DATA_BLOCK "Inputs"   // DB13
{ S7_Optimized_Access := 'FALSE' }
VERSION : 0.1
   VAR
      "BC01 run" : Bool;
      BC01_All_inv : Bool;
      "RD01 run" : Bool;
      RD01_All_inv : Bool;
      "fan RD01 run" : Bool;
      "MC03 run" : Bool;
      "MC04 run" : Bool;
      MC04_All_inv : Bool;
      "MC05 run" : Bool;
      "VS01 run" : Bool;
      VS01_All_Inv : Bool;
      "FEEDBACKMOTOR SC-12" : Bool;
      "Aux inverter RUN" : Bool;
      Aux_Inv_All : Bool;
      "MV06 Run_Opening" : Bool;
      "MV06 Run_Closing" : Bool;
      "MV05 RUN_Opening" : Bool;
      "MV05 RUN_Closing" : Bool;
      "MV02 RUN_Opening" : Bool;
      "MV02 RUN_Closing" : Bool;
      "MV03 Run_Opening" : Bool;
      "MV03 Run_Closing" : Bool;
      "MV04 RUN_Opening" : Bool;
      "MV04 RUN_Closing" : Bool;
      "FN02 Run" : Bool;
      FN02_All_Inv : Bool;
      "MV01 Run_Opening" : Bool;
      "MV01 Run_Closing" : Bool;
      "VR-01 RUN" : Bool;
      "FN01 Run" : Bool;
      FN01_All_Inv : Bool;
      "VR02 Run" : Bool;
      "CH01 Run" : Bool;
      "FN03 Run" : Bool;
      FN03_All_SoftStarter : Bool;
      "FEEDBACKMOTOR FN-06" : Bool;
      "FEEDBACKMOTOR SC-01" : Bool;
      "FEEDBACKMOTOR FN-01 FAN" : Bool;
      "FEEDBACKMOTOR LD-01" : Bool;
      "FEEDBACKMOTOR-LD-01A" : Bool;
      "FEEDBACKMOTOR SC-10" : Bool;
      "FEEDBACKMOTOR SC-11" : Bool;
      SPARE_0 : Bool;
      SPARE_1 : Bool;
      "VR03 Run" : Bool;
      "VR04 Run" : Bool;
      "VR05 Run" : Bool;
      "VR-06 RUN" : Bool;
      "FN-05 RUN" : Bool;
      Feedback_ER01 : Bool;
      "BC01 trip wire" : Bool;
      "BC01 prox" : Bool;
      "MC03 torque" : Bool;
      "MC04 torque" : Bool;
      "MC05 torque" : Bool;
      MV06_Open : Bool;
      "MV06 Close" : Bool;
      "MV05 open" : Bool;
      "MV05 Close" : Bool;
      "MV02 Open" : Bool;
      "MV02 Close" : Bool;
      "MV03 open" : Bool;
      "MV03 Close" : Bool;
      "MV04 Open" : Bool;
      "MV04 Close" : Bool;
      "MV01 Open" : Bool;
      "MV01 Close" : Bool;
      SPARE_2 : Bool;
      SPARE_3 : Bool;
      SPARE_4 : Bool;
      "FC GATE A OPEN" : Bool;
      "LIMIT SWITCH LS-02GATE A CLOSEDVALVE PV-01" : Bool;
      "PV-01 GATE B OPEN" : Bool;
      "LIMIT SWITCH LS-06GATE B CLOSEDVALVE PV-01" : Bool;
      "Selector Op Gate A PV-01" : Bool;
      "Selector Op Gate B PV-01" : Bool;
      "PV-02 EV A OPEN" : Bool;
      "PV-02 EV A CLOSE" : Bool;
      "PV-02 GATE B OPEN" : Bool;
      "PV-02 GATE B CLOSE" : Bool;
      "Selector Op Gate A PV-02" : Bool;
      "Selector Op Gate B PV-02" : Bool;
      "Deviator Open PV-03" : Bool;
      "Deviator Close PV-03" : Bool;
      "PV03 Local Selector" : Bool;
      "PV04 Open" : Bool;
      "PV04 Close" : Bool;
      "Button Open PV-0000" : Bool;
      "Low Pressure Air" : Bool;
      "BWF01 OK" : Bool;
      "BWF 01 RUN" : Bool;
      "BWF01 FAULT" : Bool;
      "min LEV BWF01" : Bool;
      "MAX LEV BWF01" : Bool;
      "BWF02 OK" : Bool;
      "BWF 02 RUN" : Bool;
      "BWF02 FAULT" : Bool;
      "min LEV BWF02" : Bool;
      "MAX LEV BWF02" : Bool;
      "APRON CONVEYOR A RUN" : Bool;
      "IMPACTOR RUN" : Bool;
      "IMPACT VIBRATIONFEEDER RUN" : Bool;
      "BELT CONVEYOR A RUN" : Bool;
      "AIR KNIFE RUN" : Bool;
      "BELT CONVEYOR B RUN" : Bool;
      "SHREDDER 1 RUN" : Bool;
      "SHREDDER VIBRATIONFEEDER RUN" : Bool;
      "BELT CONVEYOR  C RUN" : Bool;
      "ROTEX SCREEN RUN" : Bool;
      "APRON CONVEYOR B RUN" : Bool;
      "SHREDDER 2 RUN" : Bool;
      "BELT CONVEYOR  D RUN" : Bool;
      "BELT CONVEYOR E RUN" : Bool;
      "LIW SYSTEMAUTOREADER" : Bool;
      "PRIMARYSHREDDER RUN" : Bool;
      FREE : Bool;
      BWF1_INVERTER_HIGH_SPEED : Bool;
      BWF2_INVERTER_HIGH_SPEED : Bool;
      "APRON CONVEYOR A FAULT" : Bool;
      "IMPACTOR FAULT" : Bool;
      "IMPACT VIBRATIONFEEDER FAULT" : Bool;
      "BELT CONVEYOR  A FAULT" : Bool;
      "AIR KNIFE FAULT" : Bool;
      "BELT CONVEYOR B FAULT" : Bool;
      "SHREDDER 1 FAULT" : Bool;
      "SHREDDER VIBRATIONFEEDER FAULT" : Bool;
      "BELT CONVEYOR C FAULT" : Bool;
      "ROTEX SCREENFAULT" : Bool;
      "APRON CONVEYOR B FAULT" : Bool;
      "SHREDDER 2FAULT" : Bool;
      "BELT COVEYOR  D FAULT" : Bool;
      "BELT CONVEYOR  E FAULT" : Bool;
      "WEIGHTING HOPPER 2FAULT" : Bool;
      "HOPPER CONVEYOR 2FAULT" : Bool;
      "BELT CONVEYOR C FAULT_doppio!" : Bool;
      "NITROGEN TANK READY" : Bool;
      "Burner On" : Bool;
      "Brurner Lock Out" : Bool;
      "Burner ON and OK" : Bool;
      "FC GAS Chiuso" : Bool;
      "Max Pressure Gas" : Bool;
      "FC Aria chiusa" : Bool;
      "FC Aria aperta" : Bool;
      "High Flame Gas" : Bool;
      FREE_2 : Bool;
      FREE_3 : Bool;
      FREE_4 : Bool;
      FREE_5 : Bool;
      FREE_6 : Bool;
      FREE_7 : Bool;
      FREE_8 : Bool;
      FREE_9 : Bool;
      FREE_10 : Bool;
      FREE_11 : Bool;
      FREE_12 : Bool;
      FREE_13 : Bool;
      EM_OK : Bool;
      Presenza_110V : Bool;
      Tacitazione : Bool;
      Reset_allarmi : Bool;
      MV01_CHANNEL_D : Bool;
      MV01_CHANNEL_C : Bool;
      MV02_CHANNEL_D : Bool;
      MV02_CHANNEL_C : Bool;
      MV03_CHANNEL_D : Bool;
      MV03_CHANNEL_C : Bool;
      MV05_CHANNEL_D : Bool;
      MV05_CHANNEL_C : Bool;
      MV06_CHANNEL_D : Bool;
      MV06_CHANNEL_C : Bool;
      FREE_23 : Bool;
      FREE_24 : Bool;
      FREE_25 : Bool;
      FREE_26 : Bool;
      FREE_27 : Bool;
      FREE_28 : Bool;
      "PV-14 OPEN" : Bool;
      "PV-14 CLOSE" : Bool;
      "FN04 Run" : Bool;
      FN04_All_inv : Bool;
      "177T1_OK" : Bool;
      "LD-01 Minimo" : Bool;
      "LD-01 Inspection LS" : Bool;
      "LD-01 Local Button" : Bool;
      TC_04 : Word;
      TC_05 : Word;
      Flow_rate_BWF01 : Word;
      Flow_rate_BWF02 : Word;
      Level_BWF01 : Word;
      Level_BWF02 : Word;
      TC_01 : Word;
      TC_02 : Word;
      TC_03 : Word;
      TC_06 : Word;
      TC_07 : Word;
      ZT_01 : Word;
      PSH_01 : Word;
      PSH_02 : Word;
      PSH_03 : Word;
      PC_01 : Word;
      MV_04_M18A : Word;
      MV_04_MV18B : Word;
      FN02_ABSORPTION : Word;
      FN04_ABSORPTION : Word;
      RD01_ABSORBPTION : Word;
      FN01_ABSORPTION : Word;
      RO_01 : Word;
      RO_02 : Word;
      RO_03 : Word;
      RO_04 : Word;
      BR_01_RETRANSMISSION_GAS : Word;
      BR_01_RETRANSMISSION_AIR : Word;
      BR_01_MASSFLOWMETER_GAS : Word;
      BR_01_MASSFLOWMETER_AIR : Word;
   END_VAR
BEGIN
END_DATA_BLOCK

DATA_BLOCK "Output"   // DB14
{ S7_Optimized_Access := 'FALSE' }
VERSION : 0.1
   VAR
      "Start BC01" : Bool;
      "Start RD01" : Bool;
      "Start fan RD01" : Bool;
      "Start Spare Motor" : Bool;
      "Start MC04" : Bool;
      "Start MC05" : Bool;
      "Start VS01" : Bool;
      "Start SC12" : Bool;
      "Start Aux INV" : Bool;
      "Open MV06" : Bool;
      "Close MV06" : Bool;
      "Open MV05" : Bool;
      "Close MV05" : Bool;
      "Open MV02" : Bool;
      "Close MV02" : Bool;
      "Start open MV03" : Bool;
      "Start Close MV03" : Bool;
      "Open MV04" : Bool;
      "Close MV04" : Bool;
      "Start FN02" : Bool;
      "Start Open MV-01" : Bool;
      "Start Close MV-01" : Bool;
      "Start VR01" : Bool;
      "Start FN01" : Bool;
      "Start VR02" : Bool;
      "Start CH01" : Bool;
      "Start FN03" : Bool;
      "Start FN06" : Bool;
      "Start SC01" : Bool;
      "Star fan FN01" : Bool;
      "Start LD01" : Bool;
      "Start Vibrator LD-01" : Bool;
      "Start SC10" : Bool;
      "Start SC11" : Bool;
      "Start FN04" : Bool;
      "Start VR03" : Bool;
      "Start VR04" : Bool;
      "Start VR05" : Bool;
      "Start VR06" : Bool;
      "Start FN05" : Bool;
      "Start ER-01" : Bool;
      EV03 : Bool;
      "PV-01 Gate a" : Bool;
      "PV-01 GATE B EV" : Bool;
      "PV-02 GATE A EV" : Bool;
      "PV-02 GATE B EV" : Bool;
      "PV-03 GATE EV" : Bool;
      "PV-04" : Bool;
      "Abilita start chiller" : Bool;
      "START LIW FEEDER" : Bool;
      "Consenso Start BWF01" : Bool;
      "Consenso Start BWF02" : Bool;
      "Start Nitrogen" : Bool;
      "Rem. Start/Stop Burner" : Bool;
      "Temperature Interlock OK" : Bool;
      "Rst allarm Burner" : Bool;
      "Start High Flame" : Bool;
      "Forzatura scintilla" : Bool;
      Spare_30 : Bool;
      Spare_31 : Bool;
      Spare_32 : Bool;
      Spare_33 : Bool;
      Siren : Bool;
      "Blinking Ligh" : Bool;
      Spare : Bool;
      Spare_1 : Bool;
      Spare_2 : Bool;
      Spare_3 : Bool;
      Spare_4 : Bool;
      Spare_5 : Bool;
      Spare_6 : Bool;
      Spare_7 : Bool;
      Spare_8 : Bool;
      Spare_9 : Bool;
      Spare_10 : Bool;
      Spare_11 : Bool;
      Spare_12 : Bool;
      Spare_13 : Bool;
      Spare_14 : Bool;
      Spare_15 : Bool;
      Spare_16 : Bool;
      Spare_17 : Bool;
      Spare_18 : Bool;
      Spare_19 : Bool;
      Spare_20 : Bool;
      Spare_21 : Bool;
      Spare_22 : Bool;
      Spare_23 : Bool;
      Spare_24 : Bool;
      Spare_25 : Bool;
      Spare_26 : Bool;
      Spare_27 : Bool;
      Spare_28 : Bool;
      Spare_29 : Bool;
      Spare_34 : Bool;
      Spare_35 : Bool;
      "EV-11" : Bool;
      "EV-12" : Bool;
      "EV-13" : Bool;
      "EV-14" : Bool;
      "EV-15" : Bool;
      "EV-16" : Bool;
      "EV-17" : Bool;
      "EV-18" : Bool;
      "EV-19" : Bool;
      "EV-20" : Bool;
      "EV-21" : Bool;
      "EV-22" : Bool;
      "EV-23" : Bool;
      "EV-24" : Bool;
      "EV-25" : Bool;
      "EV-26" : Bool;
      "EV-27" : Bool;
      "EV-28" : Bool;
      "EV-29" : Bool;
      "EV-30" : Bool;
      "EV-31" : Bool;
      "EV-32" : Bool;
      "EV-33" : Bool;
      "EV-34" : Bool;
      "EV-35" : Bool;
      "EV-36" : Bool;
      "EV-37" : Bool;
      "EV-38" : Bool;
      "EV-39" : Bool;
      "EV-40" : Bool;
      "EV-41" : Bool;
      "EV-42" : Bool;
      "EV-43" : Bool;
      "EV-44" : Bool;
      "EV-45" : Bool;
      "EV-46" : Bool;
      "EV-47" : Bool;
      "EV-48" : Bool;
      "EV-49" : Bool;
      "EV-50" : Bool;
      "PV-14" : Bool;
      Spare_36 : Bool;
      Spare_37 : Bool;
      Spare_38 : Bool;
      Spare_39 : Bool;
      Spare_40 : Bool;
      Spare_41 : Bool;
      Spare_42 : Bool;
      "EV-51" : Bool;
      "EV-52" : Bool;
      "EV-53" : Bool;
      "EV-54" : Bool;
      "EV-55" : Bool;
      "EV-56" : Bool;
      "EV-57" : Bool;
      "EV-58" : Bool;
      "EV-59" : Bool;
      "EV-60" : Bool;
      "EV- 61" : Bool;
      "EV-62" : Bool;
      "EV-63" : Bool;
      "EV-64" : Bool;
      "EV-65" : Bool;
      "EV-66" : Bool;
      "EV-67" : Bool;
      "EV-68" : Bool;
      "EV-69" : Bool;
      "EV-70" : Bool;
      "EV-71" : Bool;
      "EV-72" : Bool;
      "EV-73" : Bool;
      "EV-74" : Bool;
      "EV-75" : Bool;
      "EV-76" : Bool;
      "EV-77" : Bool;
      "EV-78" : Bool;
      "EV-79" : Bool;
      "EV-80" : Bool;
      "EV-81" : Bool;
      "EV-82" : Bool;
      "EV-83" : Bool;
      "EV-84" : Bool;
      "EV-85" : Bool;
      "EV- 86" : Bool;
      "EV-87" : Bool;
      "EV-88" : Bool;
      "EV-89" : Bool;
      "EV-90" : Bool;
   END_VAR
BEGIN
END_DATA_BLOCK

DATA_BLOCK "RecipesDB"   // DB26
{ S7_Optimized_Access := 'FALSE' }
VERSION : 0.1
   VAR
      HMI_Index : Int;   // Recipe Currently Displayed on Editor (1...100)
      OldHmi_Idx : Int;   // Last Scan Hmi idx
      Vis_SaveUndo : Bool;   // Vsibility For Undo and Save btn
      Vis_Modify : Bool := 1;   // Vsibility For Modify btn
      Vis_LoadRecipe : Bool := 1;   // Visibility Of the load recipe btn
      Load_Recipe : Bool;   // Load Recipe In Cycle
      Save_Recipe : Bool;   // Save Recipe in Archive
      Modify_Recipe : Bool;   // Modify The Editor Displayed Recipe
      Undo_Modification : Bool;   // Undo the edits on the editor
      Active_Recipe : Int;   // Recipe Currently Used
      Recipes : Array[0..101] of "Recipe";   // 100 Records Of recipes + HMI Buffer
   END_VAR
BEGIN
   // Recipes[0] : HMI Buffer
   // Recipes[1] : Recipe #1
   // Recipes[2] : Recipe #2
   // Recipes[3] : Recipe #3
   // Recipes[4] : Recipe #4
   // Recipes[5] : Recipe #5
   // Recipes[6] : Recipe #6
   // Recipes[7] : Recipe #7
   // Recipes[8] : Recipe #8
   // Recipes[9] : Recipe #9
   // Recipes[10] : Recipe #10
   // Recipes[11] : Recipe #11
   // Recipes[12] : Recipe #12
   // Recipes[13] : Recipe #13
   // Recipes[14] : Recipe #14
   // Recipes[15] : Recipe #15
   // Recipes[16] : Recipe #16
   // Recipes[17] : Recipe #17
   // Recipes[18] : Recipe #18
   // Recipes[19] : Recipe #19
   // Recipes[20] : Recipe #20
   // Recipes[21] : Recipe #21
   // Recipes[22] : Recipe #22
   // Recipes[23] : Recipe #23
   // Recipes[24] : Recipe #24
   // Recipes[25] : Recipe #25
   // Recipes[26] : Recipe #26
   // Recipes[27] : Recipe #27
   // Recipes[28] : Recipe #28
   // Recipes[29] : Recipe #29
   // Recipes[30] : Recipe #30
   // Recipes[31] : Recipe #31
   // Recipes[32] : Recipe #32
   // Recipes[33] : Recipe #33
   // Recipes[34] : Recipe #34
   // Recipes[35] : Recipe #35
   // Recipes[36] : Recipe #36
   // Recipes[37] : Recipe #37
   // Recipes[38] : Recipe #38
   // Recipes[39] : Recipe #39
   // Recipes[40] : Recipe #40
   // Recipes[41] : Recipe #41
   // Recipes[42] : Recipe #42
   // Recipes[43] : Recipe #43
   // Recipes[44] : Recipe #44
   // Recipes[45] : Recipe #45
   // Recipes[46] : Recipe #46
   // Recipes[47] : Recipe #47
   // Recipes[48] : Recipe #48
   // Recipes[49] : Recipe #49
   // Recipes[50] : Recipe #50
   // Recipes[51] : Recipe #51
   // Recipes[52] : Recipe #52
   // Recipes[53] : Recipe #53
   // Recipes[54] : Recipe #54
   // Recipes[55] : Recipe #55
   // Recipes[56] : Recipe #56
   // Recipes[57] : Recipe #57
   // Recipes[58] : Recipe #58
   // Recipes[59] : Recipe #59
   // Recipes[60] : Recipe #60
   // Recipes[61] : Recipe #61
   // Recipes[62] : Recipe #62
   // Recipes[63] : Recipe #63
   // Recipes[64] : Recipe #64
   // Recipes[65] : Recipe #65
   // Recipes[66] : Recipe #66
   // Recipes[67] : Recipe #67
   // Recipes[68] : Recipe #68
   // Recipes[69] : Recipe #69
   // Recipes[70] : Recipe #70
   // Recipes[71] : Recipe #71
   // Recipes[72] : Recipe #72
   // Recipes[73] : Recipe #73
   // Recipes[74] : Recipe #74
   // Recipes[75] : Recipe #75
   // Recipes[76] : Recipe #76
   // Recipes[77] : Recipe #77
   // Recipes[78] : Recipe #78
   // Recipes[79] : Recipe #79
   // Recipes[80] : Recipe #80
   // Recipes[81] : Recipe #81
   // Recipes[82] : Recipe #82
   // Recipes[83] : Recipe #83
   // Recipes[84] : Recipe #84
   // Recipes[85] : Recipe #85
   // Recipes[86] : Recipe #86
   // Recipes[87] : Recipe #87
   // Recipes[88] : Recipe #88
   // Recipes[89] : Recipe #89
   // Recipes[90] : Recipe #90
   // Recipes[91] : Recipe #91
   // Recipes[92] : Recipe #92
   // Recipes[93] : Recipe #93
   // Recipes[94] : Recipe #94
   // Recipes[95] : Recipe #95
   // Recipes[96] : Recipe #96
   // Recipes[97] : Recipe #97
   // Recipes[98] : Recipe #98
   // Recipes[99] : Recipe #99
   // Recipes[100] : Recipe #100
END_DATA_BLOCK

// folder: System blocks/Program resources

DATA_BLOCK "Clock1S_simu"   // DB28
{ S7_Optimized_Access := 'TRUE' }
AUTHOR : Simatic
FAMILY : IEC
NAME : IEC_TMR
VERSION : 1.0
// stored: InstanceOfName IEC_TIMER
"IEC_TIMER"
BEGIN
END_DATA_BLOCK

DATA_BLOCK "Clock3s_simu"   // DB29
{ S7_Optimized_Access := 'TRUE' }
AUTHOR : Simatic
FAMILY : IEC
NAME : IEC_TMR
VERSION : 1.0
// stored: InstanceOfName IEC_TIMER
"IEC_TIMER"
BEGIN
END_DATA_BLOCK

DATA_BLOCK "Aux_Inv_run"   // DB31
{ S7_Optimized_Access := 'TRUE' }
AUTHOR : Simatic
FAMILY : IEC
NAME : IEC_TMR
VERSION : 1.0
// stored: InstanceOfName IEC_TIMER
"IEC_TIMER"
BEGIN
END_DATA_BLOCK

DATA_BLOCK "Er_01_Run_Rit"   // DB32
{ S7_Optimized_Access := 'TRUE' }
AUTHOR : Simatic
FAMILY : IEC
NAME : IEC_TMR
VERSION : 1.0
// stored: InstanceOfName IEC_TIMER
"IEC_TIMER"
BEGIN
END_DATA_BLOCK

DATA_BLOCK "Min_LD_01"   // DB33
{ S7_Optimized_Access := 'TRUE' }
AUTHOR : Simatic
FAMILY : IEC
NAME : IEC_TMR
VERSION : 1.0
// stored: InstanceOfName IEC_TIMER
"IEC_TIMER"
BEGIN
END_DATA_BLOCK

DATA_BLOCK "RO03_Min"   // DB34
{ S7_Optimized_Access := 'TRUE' }
AUTHOR : Simatic
FAMILY : IEC
NAME : IEC_TMR
VERSION : 1.0
// stored: InstanceOfName IEC_TIMER
"IEC_TIMER"
BEGIN
END_DATA_BLOCK

DATA_BLOCK "RO03_Max"   // DB35
{ S7_Optimized_Access := 'TRUE' }
AUTHOR : Simatic
FAMILY : IEC
NAME : IEC_TMR
VERSION : 1.0
// stored: InstanceOfName IEC_TIMER
"IEC_TIMER"
BEGIN
END_DATA_BLOCK

DATA_BLOCK "IEC_Timer_0_DB"   // DB36
{ S7_Optimized_Access := 'TRUE' }
AUTHOR : Simatic
FAMILY : IEC
NAME : IEC_TMR
VERSION : 1.0
// stored: InstanceOfName IEC_TIMER
"IEC_TIMER"
BEGIN
END_DATA_BLOCK

DATA_BLOCK "IEC_Timer_1_DB"   // DB37
{ S7_Optimized_Access := 'TRUE' }
AUTHOR : Simatic
FAMILY : IEC
NAME : IEC_TMR
VERSION : 1.0
// stored: InstanceOfName IEC_TIMER
"IEC_TIMER"
BEGIN
END_DATA_BLOCK

DATA_BLOCK "T_Reset_Startup_PV1"   // DB38
{ S7_Optimized_Access := 'TRUE' }
AUTHOR : Simatic
FAMILY : IEC
NAME : IEC_TMR
VERSION : 1.0
// stored: InstanceOfName IEC_TIMER
"IEC_TIMER"
BEGIN
END_DATA_BLOCK

DATA_BLOCK "ton_1st_step_FN01"   // DB42
{ S7_Optimized_Access := 'TRUE' }
AUTHOR : Simatic
FAMILY : IEC
NAME : IEC_TMR
VERSION : 1.0
// stored: InstanceOfName IEC_TIMER
"IEC_TIMER"
BEGIN
END_DATA_BLOCK

DATA_BLOCK "ton_2nd_step_FN01"   // DB43
{ S7_Optimized_Access := 'TRUE' }
AUTHOR : Simatic
FAMILY : IEC
NAME : IEC_TMR
VERSION : 1.0
// stored: InstanceOfName IEC_TIMER
"IEC_TIMER"
BEGIN
END_DATA_BLOCK

DATA_BLOCK "ton_3rd_step_FN01"   // DB44
{ S7_Optimized_Access := 'TRUE' }
AUTHOR : Simatic
FAMILY : IEC
NAME : IEC_TMR
VERSION : 1.0
// stored: InstanceOfName IEC_TIMER
"IEC_TIMER"
BEGIN
END_DATA_BLOCK

DATA_BLOCK "ton_4th_step_FN01"   // DB45
{ S7_Optimized_Access := 'TRUE' }
AUTHOR : Simatic
FAMILY : IEC
NAME : IEC_TMR
VERSION : 1.0
// stored: InstanceOfName IEC_TIMER
"IEC_TIMER"
BEGIN
END_DATA_BLOCK

DATA_BLOCK "ton_last_step_FN01"   // DB46
{ S7_Optimized_Access := 'TRUE' }
AUTHOR : Simatic
FAMILY : IEC
NAME : IEC_TMR
VERSION : 1.0
// stored: InstanceOfName IEC_TIMER
"IEC_TIMER"
BEGIN
END_DATA_BLOCK

DATA_BLOCK "IEC_Timer_0_DB_1"   // DB47
{ S7_Optimized_Access := 'TRUE' }
AUTHOR : Simatic
FAMILY : IEC
NAME : IEC_TMR
VERSION : 1.0
// stored: InstanceOfName IEC_TIMER
"IEC_TIMER"
BEGIN
END_DATA_BLOCK

// folder: (top level)

FUNCTION "time work motor" : Void   // FC2, LAD
{ S7_Optimized_Access := 'FALSE' }
VERSION : 0.1
   VAR_TEMP   // added for the SCL form of the ladder/FBD networks
      _w1 : Bool;
      _w2 : Bool;
   END_VAR
BEGIN

REGION Network 1: client motor 1
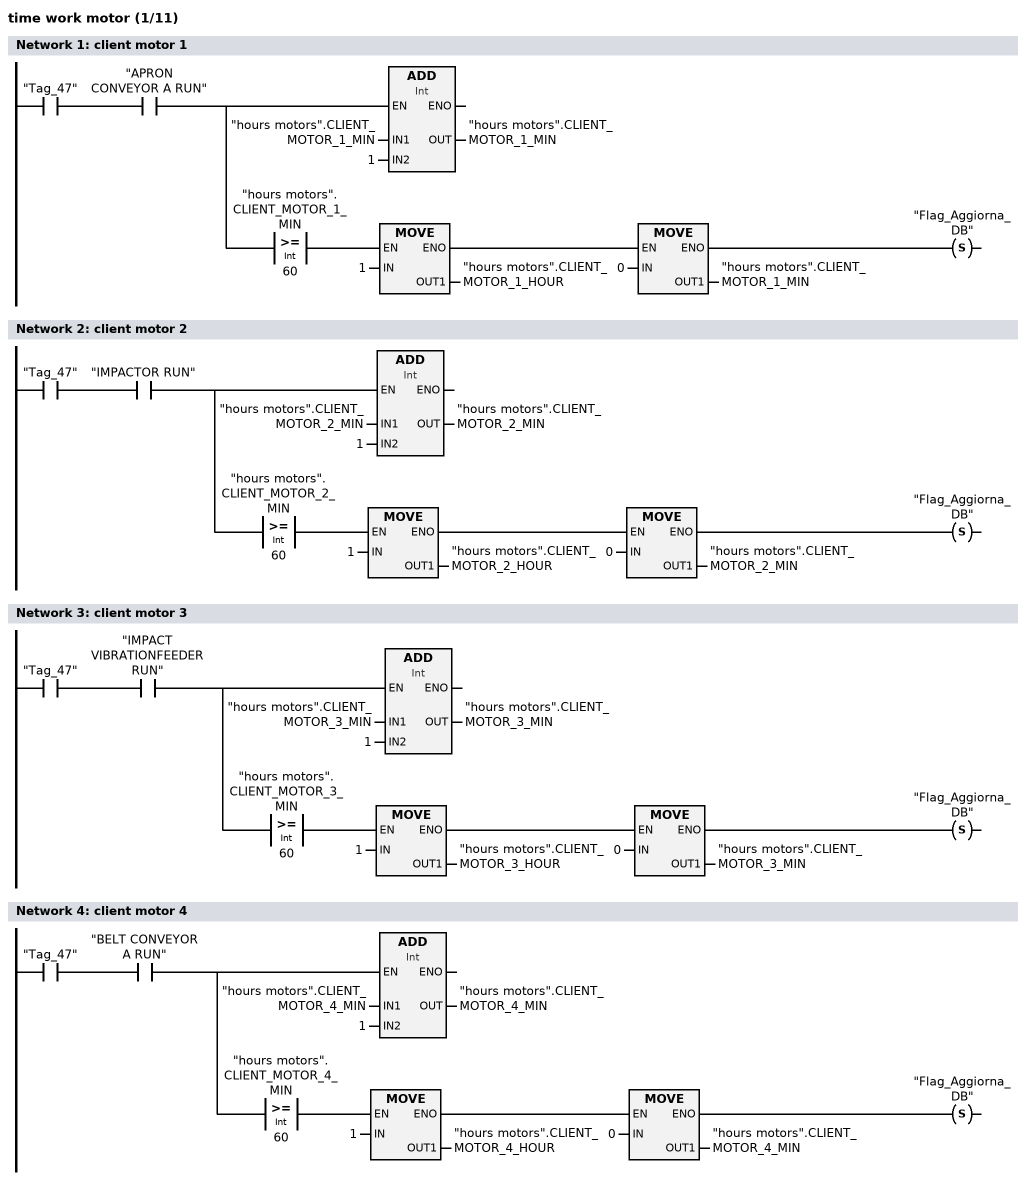
   RUNG wire#powerrail
      Contact( "Tag_47" )
      Contact( "APRON CONVEYOR A RUN" )
      wire#w1
      { S7_Templates := "SrcType := Int"; S7_GenerateENO := "TRUE" } Add(in1 := "hours motors".CLIENT_MOTOR_1_MIN, in2 := 1, out => "hours motors".CLIENT_MOTOR_1_MIN)
   END_RUNG
   RUNG wire#w1
      { S7_Templates := "SrcType := Int" } GE_Contact(in1 := "hours motors".CLIENT_MOTOR_1_MIN, in2 := 60)
      { S7_GenerateENO := "TRUE" } Move(in := 1, out1 => "hours motors".CLIENT_MOTOR_1_HOUR)
      { S7_GenerateENO := "TRUE" } Move(in := 0, out1 => "hours motors".CLIENT_MOTOR_1_MIN)
      S_Coil( "Flag_Aggiorna_DB" )
   END_RUNG
   // the same network as SCL:
   // ENO of a box is taken as its EN; it also drops when the box reports an error
   #_w1 := "Tag_47" AND "APRON CONVEYOR A RUN";
   IF #_w1 THEN "hours motors".CLIENT_MOTOR_1_MIN := "hours motors".CLIENT_MOTOR_1_MIN + 1; END_IF;
   IF #_w1 AND ("hours motors".CLIENT_MOTOR_1_MIN >= 60) THEN
       "hours motors".CLIENT_MOTOR_1_HOUR := 1;
   END_IF;
   #_w2 := #_w1 AND ("hours motors".CLIENT_MOTOR_1_MIN >= 60);
   IF #_w2 THEN
       "hours motors".CLIENT_MOTOR_1_MIN := 0;
       "Flag_Aggiorna_DB" := TRUE;
   END_IF;
END_REGION

REGION Network 2: client motor 2
   RUNG wire#powerrail
      Contact( "Tag_47" )
      Contact( "IMPACTOR RUN" )
      wire#w1
      { S7_Templates := "SrcType := Int"; S7_GenerateENO := "TRUE" } Add(in1 := "hours motors".CLIENT_MOTOR_2_MIN, in2 := 1, out => "hours motors".CLIENT_MOTOR_2_MIN)
   END_RUNG
   RUNG wire#w1
      { S7_Templates := "SrcType := Int" } GE_Contact(in1 := "hours motors".CLIENT_MOTOR_2_MIN, in2 := 60)
      { S7_GenerateENO := "TRUE" } Move(in := 1, out1 => "hours motors".CLIENT_MOTOR_2_HOUR)
      { S7_GenerateENO := "TRUE" } Move(in := 0, out1 => "hours motors".CLIENT_MOTOR_2_MIN)
      S_Coil( "Flag_Aggiorna_DB" )
   END_RUNG
   // the same network as SCL:
   // ENO of a box is taken as its EN; it also drops when the box reports an error
   #_w1 := "Tag_47" AND "IMPACTOR RUN";
   IF #_w1 THEN "hours motors".CLIENT_MOTOR_2_MIN := "hours motors".CLIENT_MOTOR_2_MIN + 1; END_IF;
   IF #_w1 AND ("hours motors".CLIENT_MOTOR_2_MIN >= 60) THEN
       "hours motors".CLIENT_MOTOR_2_HOUR := 1;
   END_IF;
   #_w2 := #_w1 AND ("hours motors".CLIENT_MOTOR_2_MIN >= 60);
   IF #_w2 THEN
       "hours motors".CLIENT_MOTOR_2_MIN := 0;
       "Flag_Aggiorna_DB" := TRUE;
   END_IF;
END_REGION

REGION Network 3: client motor 3
   RUNG wire#powerrail
      Contact( "Tag_47" )
      Contact( "IMPACT VIBRATIONFEEDER RUN" )
      wire#w1
      { S7_Templates := "SrcType := Int"; S7_GenerateENO := "TRUE" } Add(in1 := "hours motors".CLIENT_MOTOR_3_MIN, in2 := 1, out => "hours motors".CLIENT_MOTOR_3_MIN)
   END_RUNG
   RUNG wire#w1
      { S7_Templates := "SrcType := Int" } GE_Contact(in1 := "hours motors".CLIENT_MOTOR_3_MIN, in2 := 60)
      { S7_GenerateENO := "TRUE" } Move(in := 1, out1 => "hours motors".CLIENT_MOTOR_3_HOUR)
      { S7_GenerateENO := "TRUE" } Move(in := 0, out1 => "hours motors".CLIENT_MOTOR_3_MIN)
      S_Coil( "Flag_Aggiorna_DB" )
   END_RUNG
   // the same network as SCL:
   // ENO of a box is taken as its EN; it also drops when the box reports an error
   #_w1 := "Tag_47" AND "IMPACT VIBRATIONFEEDER RUN";
   IF #_w1 THEN "hours motors".CLIENT_MOTOR_3_MIN := "hours motors".CLIENT_MOTOR_3_MIN + 1; END_IF;
   IF #_w1 AND ("hours motors".CLIENT_MOTOR_3_MIN >= 60) THEN
       "hours motors".CLIENT_MOTOR_3_HOUR := 1;
   END_IF;
   #_w2 := #_w1 AND ("hours motors".CLIENT_MOTOR_3_MIN >= 60);
   IF #_w2 THEN
       "hours motors".CLIENT_MOTOR_3_MIN := 0;
       "Flag_Aggiorna_DB" := TRUE;
   END_IF;
END_REGION

REGION Network 4: client motor 4
   RUNG wire#powerrail
      Contact( "Tag_47" )
      Contact( "BELT CONVEYOR A RUN" )
      wire#w1
      { S7_Templates := "SrcType := Int"; S7_GenerateENO := "TRUE" } Add(in1 := "hours motors".CLIENT_MOTOR_4_MIN, in2 := 1, out => "hours motors".CLIENT_MOTOR_4_MIN)
   END_RUNG
   RUNG wire#w1
      { S7_Templates := "SrcType := Int" } GE_Contact(in1 := "hours motors".CLIENT_MOTOR_4_MIN, in2 := 60)
      { S7_GenerateENO := "TRUE" } Move(in := 1, out1 => "hours motors".CLIENT_MOTOR_4_HOUR)
      { S7_GenerateENO := "TRUE" } Move(in := 0, out1 => "hours motors".CLIENT_MOTOR_4_MIN)
      S_Coil( "Flag_Aggiorna_DB" )
   END_RUNG
   // the same network as SCL:
   // ENO of a box is taken as its EN; it also drops when the box reports an error
   #_w1 := "Tag_47" AND "BELT CONVEYOR A RUN";
   IF #_w1 THEN "hours motors".CLIENT_MOTOR_4_MIN := "hours motors".CLIENT_MOTOR_4_MIN + 1; END_IF;
   IF #_w1 AND ("hours motors".CLIENT_MOTOR_4_MIN >= 60) THEN
       "hours motors".CLIENT_MOTOR_4_HOUR := 1;
   END_IF;
   #_w2 := #_w1 AND ("hours motors".CLIENT_MOTOR_4_MIN >= 60);
   IF #_w2 THEN
       "hours motors".CLIENT_MOTOR_4_MIN := 0;
       "Flag_Aggiorna_DB" := TRUE;
   END_IF;
END_REGION

REGION Network 5: client motor 5
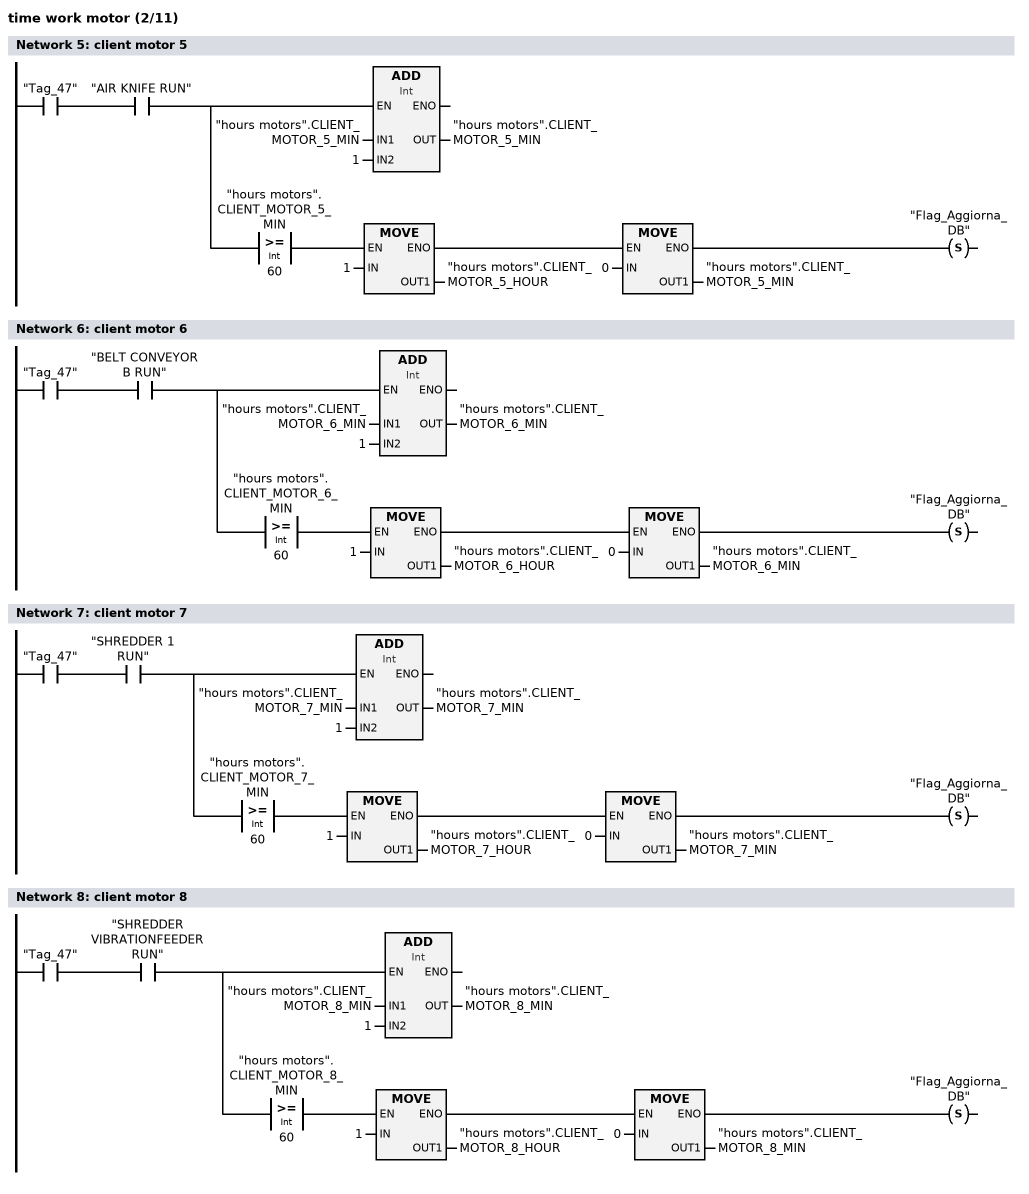
   RUNG wire#powerrail
      Contact( "Tag_47" )
      Contact( "AIR KNIFE RUN" )
      wire#w1
      { S7_Templates := "SrcType := Int"; S7_GenerateENO := "TRUE" } Add(in1 := "hours motors".CLIENT_MOTOR_5_MIN, in2 := 1, out => "hours motors".CLIENT_MOTOR_5_MIN)
   END_RUNG
   RUNG wire#w1
      { S7_Templates := "SrcType := Int" } GE_Contact(in1 := "hours motors".CLIENT_MOTOR_5_MIN, in2 := 60)
      { S7_GenerateENO := "TRUE" } Move(in := 1, out1 => "hours motors".CLIENT_MOTOR_5_HOUR)
      { S7_GenerateENO := "TRUE" } Move(in := 0, out1 => "hours motors".CLIENT_MOTOR_5_MIN)
      S_Coil( "Flag_Aggiorna_DB" )
   END_RUNG
   // the same network as SCL:
   // ENO of a box is taken as its EN; it also drops when the box reports an error
   #_w1 := "Tag_47" AND "AIR KNIFE RUN";
   IF #_w1 THEN "hours motors".CLIENT_MOTOR_5_MIN := "hours motors".CLIENT_MOTOR_5_MIN + 1; END_IF;
   IF #_w1 AND ("hours motors".CLIENT_MOTOR_5_MIN >= 60) THEN
       "hours motors".CLIENT_MOTOR_5_HOUR := 1;
   END_IF;
   #_w2 := #_w1 AND ("hours motors".CLIENT_MOTOR_5_MIN >= 60);
   IF #_w2 THEN
       "hours motors".CLIENT_MOTOR_5_MIN := 0;
       "Flag_Aggiorna_DB" := TRUE;
   END_IF;
END_REGION

REGION Network 6: client motor 6
   RUNG wire#powerrail
      Contact( "Tag_47" )
      Contact( "BELT CONVEYOR B RUN" )
      wire#w1
      { S7_Templates := "SrcType := Int"; S7_GenerateENO := "TRUE" } Add(in1 := "hours motors".CLIENT_MOTOR_6_MIN, in2 := 1, out => "hours motors".CLIENT_MOTOR_6_MIN)
   END_RUNG
   RUNG wire#w1
      { S7_Templates := "SrcType := Int" } GE_Contact(in1 := "hours motors".CLIENT_MOTOR_6_MIN, in2 := 60)
      { S7_GenerateENO := "TRUE" } Move(in := 1, out1 => "hours motors".CLIENT_MOTOR_6_HOUR)
      { S7_GenerateENO := "TRUE" } Move(in := 0, out1 => "hours motors".CLIENT_MOTOR_6_MIN)
      S_Coil( "Flag_Aggiorna_DB" )
   END_RUNG
   // the same network as SCL:
   // ENO of a box is taken as its EN; it also drops when the box reports an error
   #_w1 := "Tag_47" AND "BELT CONVEYOR B RUN";
   IF #_w1 THEN "hours motors".CLIENT_MOTOR_6_MIN := "hours motors".CLIENT_MOTOR_6_MIN + 1; END_IF;
   IF #_w1 AND ("hours motors".CLIENT_MOTOR_6_MIN >= 60) THEN
       "hours motors".CLIENT_MOTOR_6_HOUR := 1;
   END_IF;
   #_w2 := #_w1 AND ("hours motors".CLIENT_MOTOR_6_MIN >= 60);
   IF #_w2 THEN
       "hours motors".CLIENT_MOTOR_6_MIN := 0;
       "Flag_Aggiorna_DB" := TRUE;
   END_IF;
END_REGION

REGION Network 7: client motor 7
   RUNG wire#powerrail
      Contact( "Tag_47" )
      Contact( "SHREDDER 1 RUN" )
      wire#w1
      { S7_Templates := "SrcType := Int"; S7_GenerateENO := "TRUE" } Add(in1 := "hours motors".CLIENT_MOTOR_7_MIN, in2 := 1, out => "hours motors".CLIENT_MOTOR_7_MIN)
   END_RUNG
   RUNG wire#w1
      { S7_Templates := "SrcType := Int" } GE_Contact(in1 := "hours motors".CLIENT_MOTOR_7_MIN, in2 := 60)
      { S7_GenerateENO := "TRUE" } Move(in := 1, out1 => "hours motors".CLIENT_MOTOR_7_HOUR)
      { S7_GenerateENO := "TRUE" } Move(in := 0, out1 => "hours motors".CLIENT_MOTOR_7_MIN)
      S_Coil( "Flag_Aggiorna_DB" )
   END_RUNG
   // the same network as SCL:
   // ENO of a box is taken as its EN; it also drops when the box reports an error
   #_w1 := "Tag_47" AND "SHREDDER 1 RUN";
   IF #_w1 THEN "hours motors".CLIENT_MOTOR_7_MIN := "hours motors".CLIENT_MOTOR_7_MIN + 1; END_IF;
   IF #_w1 AND ("hours motors".CLIENT_MOTOR_7_MIN >= 60) THEN
       "hours motors".CLIENT_MOTOR_7_HOUR := 1;
   END_IF;
   #_w2 := #_w1 AND ("hours motors".CLIENT_MOTOR_7_MIN >= 60);
   IF #_w2 THEN
       "hours motors".CLIENT_MOTOR_7_MIN := 0;
       "Flag_Aggiorna_DB" := TRUE;
   END_IF;
END_REGION

REGION Network 8: client motor 8
   RUNG wire#powerrail
      Contact( "Tag_47" )
      Contact( "SHREDDER VIBRATIONFEEDER RUN" )
      wire#w1
      { S7_Templates := "SrcType := Int"; S7_GenerateENO := "TRUE" } Add(in1 := "hours motors".CLIENT_MOTOR_8_MIN, in2 := 1, out => "hours motors".CLIENT_MOTOR_8_MIN)
   END_RUNG
   RUNG wire#w1
      { S7_Templates := "SrcType := Int" } GE_Contact(in1 := "hours motors".CLIENT_MOTOR_8_MIN, in2 := 60)
      { S7_GenerateENO := "TRUE" } Move(in := 1, out1 => "hours motors".CLIENT_MOTOR_8_HOUR)
      { S7_GenerateENO := "TRUE" } Move(in := 0, out1 => "hours motors".CLIENT_MOTOR_8_MIN)
      S_Coil( "Flag_Aggiorna_DB" )
   END_RUNG
   // the same network as SCL:
   // ENO of a box is taken as its EN; it also drops when the box reports an error
   #_w1 := "Tag_47" AND "SHREDDER VIBRATIONFEEDER RUN";
   IF #_w1 THEN "hours motors".CLIENT_MOTOR_8_MIN := "hours motors".CLIENT_MOTOR_8_MIN + 1; END_IF;
   IF #_w1 AND ("hours motors".CLIENT_MOTOR_8_MIN >= 60) THEN
       "hours motors".CLIENT_MOTOR_8_HOUR := 1;
   END_IF;
   #_w2 := #_w1 AND ("hours motors".CLIENT_MOTOR_8_MIN >= 60);
   IF #_w2 THEN
       "hours motors".CLIENT_MOTOR_8_MIN := 0;
       "Flag_Aggiorna_DB" := TRUE;
   END_IF;
END_REGION

REGION Network 9: client motor 9
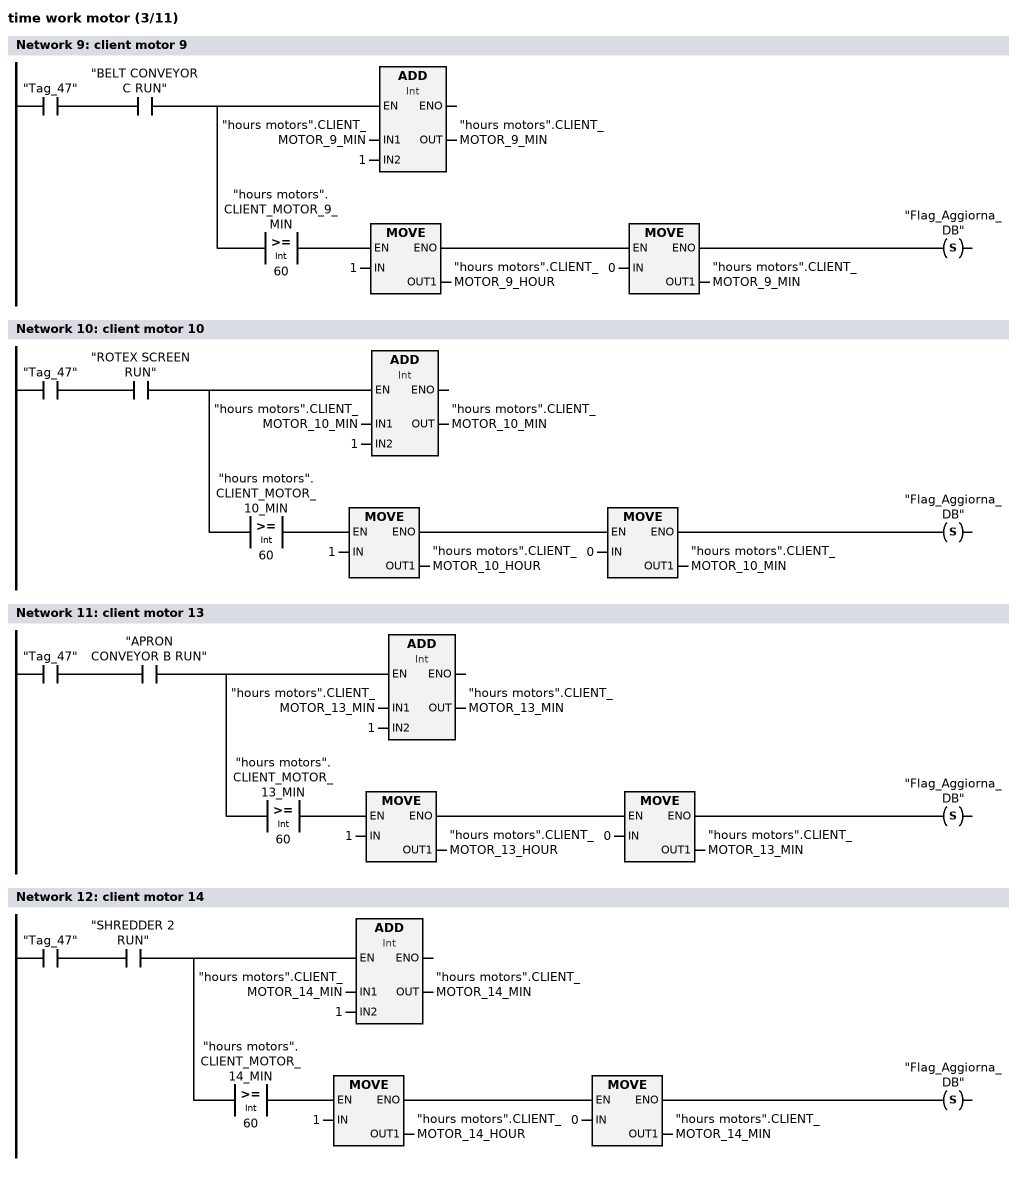
   RUNG wire#powerrail
      Contact( "Tag_47" )
      Contact( "BELT CONVEYOR  C RUN" )
      wire#w1
      { S7_Templates := "SrcType := Int"; S7_GenerateENO := "TRUE" } Add(in1 := "hours motors".CLIENT_MOTOR_9_MIN, in2 := 1, out => "hours motors".CLIENT_MOTOR_9_MIN)
   END_RUNG
   RUNG wire#w1
      { S7_Templates := "SrcType := Int" } GE_Contact(in1 := "hours motors".CLIENT_MOTOR_9_MIN, in2 := 60)
      { S7_GenerateENO := "TRUE" } Move(in := 1, out1 => "hours motors".CLIENT_MOTOR_9_HOUR)
      { S7_GenerateENO := "TRUE" } Move(in := 0, out1 => "hours motors".CLIENT_MOTOR_9_MIN)
      S_Coil( "Flag_Aggiorna_DB" )
   END_RUNG
   // the same network as SCL:
   // ENO of a box is taken as its EN; it also drops when the box reports an error
   #_w1 := "Tag_47" AND "BELT CONVEYOR  C RUN";
   IF #_w1 THEN "hours motors".CLIENT_MOTOR_9_MIN := "hours motors".CLIENT_MOTOR_9_MIN + 1; END_IF;
   IF #_w1 AND ("hours motors".CLIENT_MOTOR_9_MIN >= 60) THEN
       "hours motors".CLIENT_MOTOR_9_HOUR := 1;
   END_IF;
   #_w2 := #_w1 AND ("hours motors".CLIENT_MOTOR_9_MIN >= 60);
   IF #_w2 THEN
       "hours motors".CLIENT_MOTOR_9_MIN := 0;
       "Flag_Aggiorna_DB" := TRUE;
   END_IF;
END_REGION

REGION Network 10: client motor 10
   RUNG wire#powerrail
      Contact( "Tag_47" )
      Contact( "ROTEX SCREEN RUN" )
      wire#w1
      { S7_Templates := "SrcType := Int"; S7_GenerateENO := "TRUE" } Add(in1 := "hours motors".CLIENT_MOTOR_10_MIN, in2 := 1, out => "hours motors".CLIENT_MOTOR_10_MIN)
   END_RUNG
   RUNG wire#w1
      { S7_Templates := "SrcType := Int" } GE_Contact(in1 := "hours motors".CLIENT_MOTOR_10_MIN, in2 := 60)
      { S7_GenerateENO := "TRUE" } Move(in := 1, out1 => "hours motors".CLIENT_MOTOR_10_HOUR)
      { S7_GenerateENO := "TRUE" } Move(in := 0, out1 => "hours motors".CLIENT_MOTOR_10_MIN)
      S_Coil( "Flag_Aggiorna_DB" )
   END_RUNG
   // the same network as SCL:
   // ENO of a box is taken as its EN; it also drops when the box reports an error
   #_w1 := "Tag_47" AND "ROTEX SCREEN RUN";
   IF #_w1 THEN "hours motors".CLIENT_MOTOR_10_MIN := "hours motors".CLIENT_MOTOR_10_MIN + 1; END_IF;
   IF #_w1 AND ("hours motors".CLIENT_MOTOR_10_MIN >= 60) THEN
       "hours motors".CLIENT_MOTOR_10_HOUR := 1;
   END_IF;
   #_w2 := #_w1 AND ("hours motors".CLIENT_MOTOR_10_MIN >= 60);
   IF #_w2 THEN
       "hours motors".CLIENT_MOTOR_10_MIN := 0;
       "Flag_Aggiorna_DB" := TRUE;
   END_IF;
END_REGION

REGION Network 11: client motor 13
   RUNG wire#powerrail
      Contact( "Tag_47" )
      Contact( "APRON CONVEYOR B RUN" )
      wire#w1
      { S7_Templates := "SrcType := Int"; S7_GenerateENO := "TRUE" } Add(in1 := "hours motors".CLIENT_MOTOR_13_MIN, in2 := 1, out => "hours motors".CLIENT_MOTOR_13_MIN)
   END_RUNG
   RUNG wire#w1
      { S7_Templates := "SrcType := Int" } GE_Contact(in1 := "hours motors".CLIENT_MOTOR_13_MIN, in2 := 60)
      { S7_GenerateENO := "TRUE" } Move(in := 1, out1 => "hours motors".CLIENT_MOTOR_13_HOUR)
      { S7_GenerateENO := "TRUE" } Move(in := 0, out1 => "hours motors".CLIENT_MOTOR_13_MIN)
      S_Coil( "Flag_Aggiorna_DB" )
   END_RUNG
   // the same network as SCL:
   // ENO of a box is taken as its EN; it also drops when the box reports an error
   #_w1 := "Tag_47" AND "APRON CONVEYOR B RUN";
   IF #_w1 THEN "hours motors".CLIENT_MOTOR_13_MIN := "hours motors".CLIENT_MOTOR_13_MIN + 1; END_IF;
   IF #_w1 AND ("hours motors".CLIENT_MOTOR_13_MIN >= 60) THEN
       "hours motors".CLIENT_MOTOR_13_HOUR := 1;
   END_IF;
   #_w2 := #_w1 AND ("hours motors".CLIENT_MOTOR_13_MIN >= 60);
   IF #_w2 THEN
       "hours motors".CLIENT_MOTOR_13_MIN := 0;
       "Flag_Aggiorna_DB" := TRUE;
   END_IF;
END_REGION

REGION Network 12: client motor 14
   RUNG wire#powerrail
      Contact( "Tag_47" )
      Contact( "SHREDDER 2 RUN" )
      wire#w1
      { S7_Templates := "SrcType := Int"; S7_GenerateENO := "TRUE" } Add(in1 := "hours motors".CLIENT_MOTOR_14_MIN, in2 := 1, out => "hours motors".CLIENT_MOTOR_14_MIN)
   END_RUNG
   RUNG wire#w1
      { S7_Templates := "SrcType := Int" } GE_Contact(in1 := "hours motors".CLIENT_MOTOR_14_MIN, in2 := 60)
      { S7_GenerateENO := "TRUE" } Move(in := 1, out1 => "hours motors".CLIENT_MOTOR_14_HOUR)
      { S7_GenerateENO := "TRUE" } Move(in := 0, out1 => "hours motors".CLIENT_MOTOR_14_MIN)
      S_Coil( "Flag_Aggiorna_DB" )
   END_RUNG
   // the same network as SCL:
   // ENO of a box is taken as its EN; it also drops when the box reports an error
   #_w1 := "Tag_47" AND "SHREDDER 2 RUN";
   IF #_w1 THEN "hours motors".CLIENT_MOTOR_14_MIN := "hours motors".CLIENT_MOTOR_14_MIN + 1; END_IF;
   IF #_w1 AND ("hours motors".CLIENT_MOTOR_14_MIN >= 60) THEN
       "hours motors".CLIENT_MOTOR_14_HOUR := 1;
   END_IF;
   #_w2 := #_w1 AND ("hours motors".CLIENT_MOTOR_14_MIN >= 60);
   IF #_w2 THEN
       "hours motors".CLIENT_MOTOR_14_MIN := 0;
       "Flag_Aggiorna_DB" := TRUE;
   END_IF;
END_REGION

REGION Network 13: client motor 15
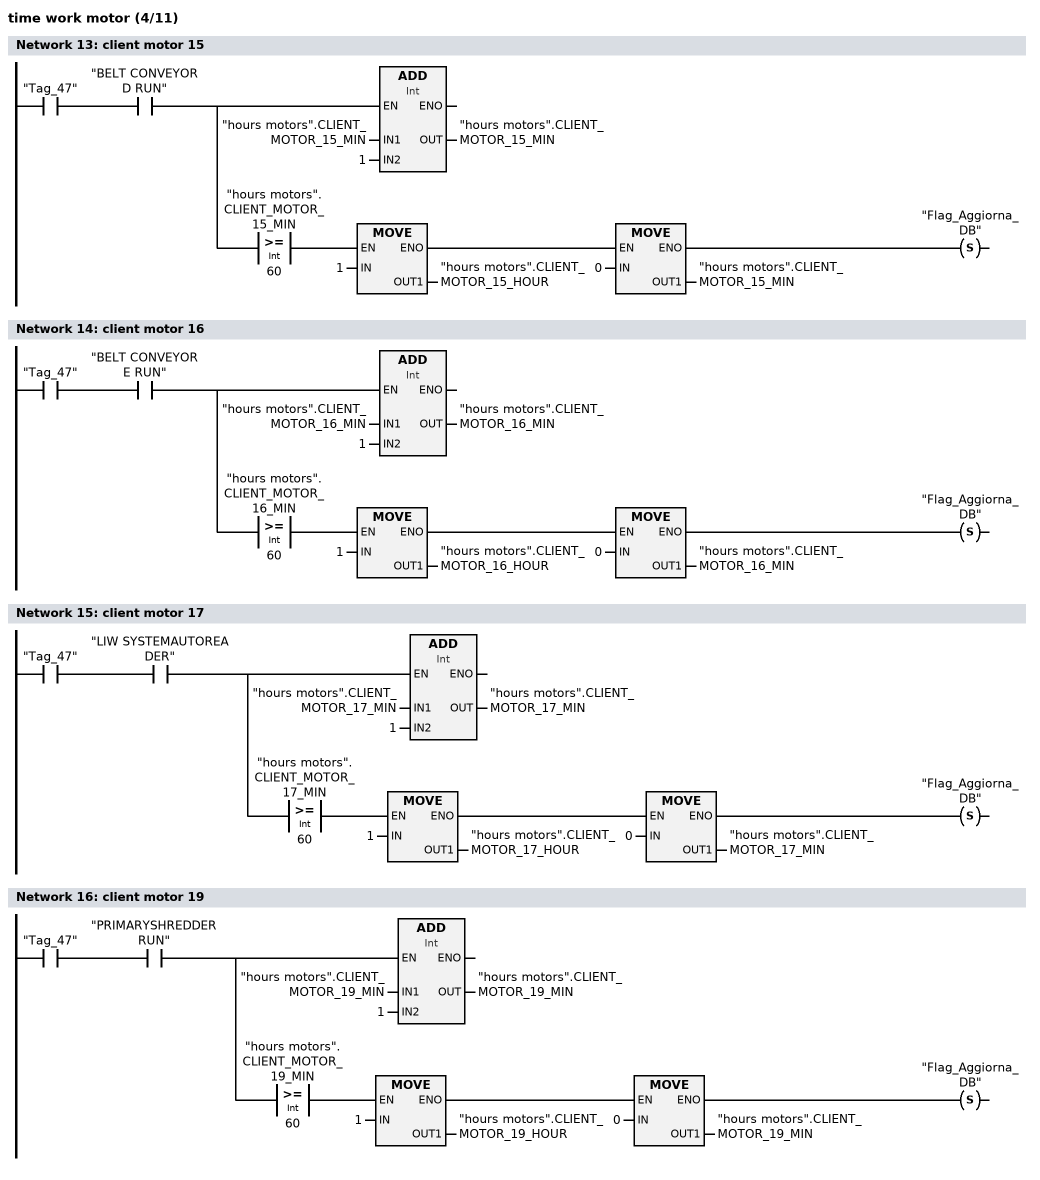
   RUNG wire#powerrail
      Contact( "Tag_47" )
      Contact( "BELT CONVEYOR  D RUN" )
      wire#w1
      { S7_Templates := "SrcType := Int"; S7_GenerateENO := "TRUE" } Add(in1 := "hours motors".CLIENT_MOTOR_15_MIN, in2 := 1, out => "hours motors".CLIENT_MOTOR_15_MIN)
   END_RUNG
   RUNG wire#w1
      { S7_Templates := "SrcType := Int" } GE_Contact(in1 := "hours motors".CLIENT_MOTOR_15_MIN, in2 := 60)
      { S7_GenerateENO := "TRUE" } Move(in := 1, out1 => "hours motors".CLIENT_MOTOR_15_HOUR)
      { S7_GenerateENO := "TRUE" } Move(in := 0, out1 => "hours motors".CLIENT_MOTOR_15_MIN)
      S_Coil( "Flag_Aggiorna_DB" )
   END_RUNG
   // the same network as SCL:
   // ENO of a box is taken as its EN; it also drops when the box reports an error
   #_w1 := "Tag_47" AND "BELT CONVEYOR  D RUN";
   IF #_w1 THEN "hours motors".CLIENT_MOTOR_15_MIN := "hours motors".CLIENT_MOTOR_15_MIN + 1; END_IF;
   IF #_w1 AND ("hours motors".CLIENT_MOTOR_15_MIN >= 60) THEN
       "hours motors".CLIENT_MOTOR_15_HOUR := 1;
   END_IF;
   #_w2 := #_w1 AND ("hours motors".CLIENT_MOTOR_15_MIN >= 60);
   IF #_w2 THEN
       "hours motors".CLIENT_MOTOR_15_MIN := 0;
       "Flag_Aggiorna_DB" := TRUE;
   END_IF;
END_REGION

REGION Network 14: client motor 16
   RUNG wire#powerrail
      Contact( "Tag_47" )
      Contact( "BELT CONVEYOR E RUN" )
      wire#w1
      { S7_Templates := "SrcType := Int"; S7_GenerateENO := "TRUE" } Add(in1 := "hours motors".CLIENT_MOTOR_16_MIN, in2 := 1, out => "hours motors".CLIENT_MOTOR_16_MIN)
   END_RUNG
   RUNG wire#w1
      { S7_Templates := "SrcType := Int" } GE_Contact(in1 := "hours motors".CLIENT_MOTOR_16_MIN, in2 := 60)
      { S7_GenerateENO := "TRUE" } Move(in := 1, out1 => "hours motors".CLIENT_MOTOR_16_HOUR)
      { S7_GenerateENO := "TRUE" } Move(in := 0, out1 => "hours motors".CLIENT_MOTOR_16_MIN)
      S_Coil( "Flag_Aggiorna_DB" )
   END_RUNG
   // the same network as SCL:
   // ENO of a box is taken as its EN; it also drops when the box reports an error
   #_w1 := "Tag_47" AND "BELT CONVEYOR E RUN";
   IF #_w1 THEN "hours motors".CLIENT_MOTOR_16_MIN := "hours motors".CLIENT_MOTOR_16_MIN + 1; END_IF;
   IF #_w1 AND ("hours motors".CLIENT_MOTOR_16_MIN >= 60) THEN
       "hours motors".CLIENT_MOTOR_16_HOUR := 1;
   END_IF;
   #_w2 := #_w1 AND ("hours motors".CLIENT_MOTOR_16_MIN >= 60);
   IF #_w2 THEN
       "hours motors".CLIENT_MOTOR_16_MIN := 0;
       "Flag_Aggiorna_DB" := TRUE;
   END_IF;
END_REGION

REGION Network 15: client motor 17
   RUNG wire#powerrail
      Contact( "Tag_47" )
      Contact( "LIW SYSTEMAUTOREADER" )
      wire#w1
      { S7_Templates := "SrcType := Int"; S7_GenerateENO := "TRUE" } Add(in1 := "hours motors".CLIENT_MOTOR_17_MIN, in2 := 1, out => "hours motors".CLIENT_MOTOR_17_MIN)
   END_RUNG
   RUNG wire#w1
      { S7_Templates := "SrcType := Int" } GE_Contact(in1 := "hours motors".CLIENT_MOTOR_17_MIN, in2 := 60)
      { S7_GenerateENO := "TRUE" } Move(in := 1, out1 => "hours motors".CLIENT_MOTOR_17_HOUR)
      { S7_GenerateENO := "TRUE" } Move(in := 0, out1 => "hours motors".CLIENT_MOTOR_17_MIN)
      S_Coil( "Flag_Aggiorna_DB" )
   END_RUNG
   // the same network as SCL:
   // ENO of a box is taken as its EN; it also drops when the box reports an error
   #_w1 := "Tag_47" AND "LIW SYSTEMAUTOREADER";
   IF #_w1 THEN "hours motors".CLIENT_MOTOR_17_MIN := "hours motors".CLIENT_MOTOR_17_MIN + 1; END_IF;
   IF #_w1 AND ("hours motors".CLIENT_MOTOR_17_MIN >= 60) THEN
       "hours motors".CLIENT_MOTOR_17_HOUR := 1;
   END_IF;
   #_w2 := #_w1 AND ("hours motors".CLIENT_MOTOR_17_MIN >= 60);
   IF #_w2 THEN
       "hours motors".CLIENT_MOTOR_17_MIN := 0;
       "Flag_Aggiorna_DB" := TRUE;
   END_IF;
END_REGION

REGION Network 16: client motor 19
   RUNG wire#powerrail
      Contact( "Tag_47" )
      Contact( "PRIMARYSHREDDER RUN" )
      wire#w1
      { S7_Templates := "SrcType := Int"; S7_GenerateENO := "TRUE" } Add(in1 := "hours motors".CLIENT_MOTOR_19_MIN, in2 := 1, out => "hours motors".CLIENT_MOTOR_19_MIN)
   END_RUNG
   RUNG wire#w1
      { S7_Templates := "SrcType := Int" } GE_Contact(in1 := "hours motors".CLIENT_MOTOR_19_MIN, in2 := 60)
      { S7_GenerateENO := "TRUE" } Move(in := 1, out1 => "hours motors".CLIENT_MOTOR_19_HOUR)
      { S7_GenerateENO := "TRUE" } Move(in := 0, out1 => "hours motors".CLIENT_MOTOR_19_MIN)
      S_Coil( "Flag_Aggiorna_DB" )
   END_RUNG
   // the same network as SCL:
   // ENO of a box is taken as its EN; it also drops when the box reports an error
   #_w1 := "Tag_47" AND "PRIMARYSHREDDER RUN";
   IF #_w1 THEN "hours motors".CLIENT_MOTOR_19_MIN := "hours motors".CLIENT_MOTOR_19_MIN + 1; END_IF;
   IF #_w1 AND ("hours motors".CLIENT_MOTOR_19_MIN >= 60) THEN
       "hours motors".CLIENT_MOTOR_19_HOUR := 1;
   END_IF;
   #_w2 := #_w1 AND ("hours motors".CLIENT_MOTOR_19_MIN >= 60);
   IF #_w2 THEN
       "hours motors".CLIENT_MOTOR_19_MIN := 0;
       "Flag_Aggiorna_DB" := TRUE;
   END_IF;
END_REGION

REGION Network 17: BC-01
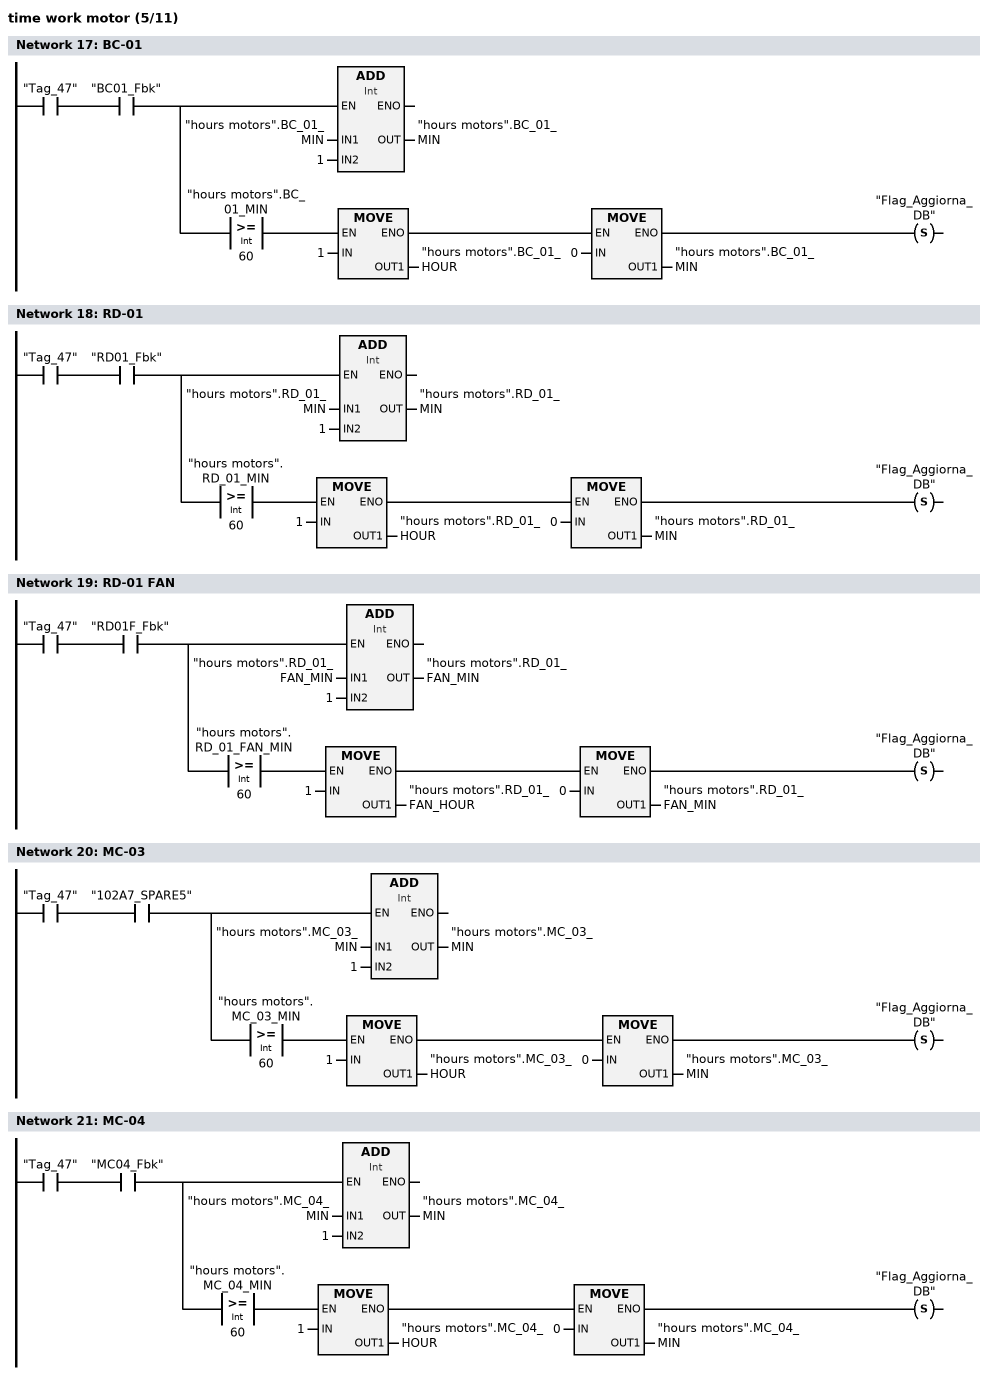
   RUNG wire#powerrail
      Contact( "Tag_47" )
      Contact( "BC01_Fbk" )
      wire#w1
      { S7_Templates := "SrcType := Int"; S7_GenerateENO := "TRUE" } Add(in1 := "hours motors".BC_01_MIN, in2 := 1, out => "hours motors".BC_01_MIN)
   END_RUNG
   RUNG wire#w1
      { S7_Templates := "SrcType := Int" } GE_Contact(in1 := "hours motors".BC_01_MIN, in2 := 60)
      { S7_GenerateENO := "TRUE" } Move(in := 1, out1 => "hours motors".BC_01_HOUR)
      { S7_GenerateENO := "TRUE" } Move(in := 0, out1 => "hours motors".BC_01_MIN)
      S_Coil( "Flag_Aggiorna_DB" )
   END_RUNG
   // the same network as SCL:
   // ENO of a box is taken as its EN; it also drops when the box reports an error
   #_w1 := "Tag_47" AND "BC01_Fbk";
   IF #_w1 THEN "hours motors".BC_01_MIN := "hours motors".BC_01_MIN + 1; END_IF;
   IF #_w1 AND ("hours motors".BC_01_MIN >= 60) THEN "hours motors".BC_01_HOUR := 1; END_IF;
   #_w2 := #_w1 AND ("hours motors".BC_01_MIN >= 60);
   IF #_w2 THEN
       "hours motors".BC_01_MIN := 0;
       "Flag_Aggiorna_DB" := TRUE;
   END_IF;
END_REGION

REGION Network 18: RD-01
   RUNG wire#powerrail
      Contact( "Tag_47" )
      Contact( "RD01_Fbk" )
      wire#w1
      { S7_Templates := "SrcType := Int"; S7_GenerateENO := "TRUE" } Add(in1 := "hours motors".RD_01_MIN, in2 := 1, out => "hours motors".RD_01_MIN)
   END_RUNG
   RUNG wire#w1
      { S7_Templates := "SrcType := Int" } GE_Contact(in1 := "hours motors".RD_01_MIN, in2 := 60)
      { S7_GenerateENO := "TRUE" } Move(in := 1, out1 => "hours motors".RD_01_HOUR)
      { S7_GenerateENO := "TRUE" } Move(in := 0, out1 => "hours motors".RD_01_MIN)
      S_Coil( "Flag_Aggiorna_DB" )
   END_RUNG
   // the same network as SCL:
   // ENO of a box is taken as its EN; it also drops when the box reports an error
   #_w1 := "Tag_47" AND "RD01_Fbk";
   IF #_w1 THEN "hours motors".RD_01_MIN := "hours motors".RD_01_MIN + 1; END_IF;
   IF #_w1 AND ("hours motors".RD_01_MIN >= 60) THEN "hours motors".RD_01_HOUR := 1; END_IF;
   #_w2 := #_w1 AND ("hours motors".RD_01_MIN >= 60);
   IF #_w2 THEN
       "hours motors".RD_01_MIN := 0;
       "Flag_Aggiorna_DB" := TRUE;
   END_IF;
END_REGION

REGION Network 19: RD-01 FAN
   RUNG wire#powerrail
      Contact( "Tag_47" )
      Contact( "RD01F_Fbk" )
      wire#w1
      { S7_Templates := "SrcType := Int"; S7_GenerateENO := "TRUE" } Add(in1 := "hours motors".RD_01_FAN_MIN, in2 := 1, out => "hours motors".RD_01_FAN_MIN)
   END_RUNG
   RUNG wire#w1
      { S7_Templates := "SrcType := Int" } GE_Contact(in1 := "hours motors".RD_01_FAN_MIN, in2 := 60)
      { S7_GenerateENO := "TRUE" } Move(in := 1, out1 => "hours motors".RD_01_FAN_HOUR)
      { S7_GenerateENO := "TRUE" } Move(in := 0, out1 => "hours motors".RD_01_FAN_MIN)
      S_Coil( "Flag_Aggiorna_DB" )
   END_RUNG
   // the same network as SCL:
   // ENO of a box is taken as its EN; it also drops when the box reports an error
   #_w1 := "Tag_47" AND "RD01F_Fbk";
   IF #_w1 THEN "hours motors".RD_01_FAN_MIN := "hours motors".RD_01_FAN_MIN + 1; END_IF;
   IF #_w1 AND ("hours motors".RD_01_FAN_MIN >= 60) THEN "hours motors".RD_01_FAN_HOUR := 1; END_IF;
   #_w2 := #_w1 AND ("hours motors".RD_01_FAN_MIN >= 60);
   IF #_w2 THEN
       "hours motors".RD_01_FAN_MIN := 0;
       "Flag_Aggiorna_DB" := TRUE;
   END_IF;
END_REGION

REGION Network 20: MC-03
   RUNG wire#powerrail
      Contact( "Tag_47" )
      Contact( "102A7_SPARE5" )
      wire#w1
      { S7_Templates := "SrcType := Int"; S7_GenerateENO := "TRUE" } Add(in1 := "hours motors".MC_03_MIN, in2 := 1, out => "hours motors".MC_03_MIN)
   END_RUNG
   RUNG wire#w1
      { S7_Templates := "SrcType := Int" } GE_Contact(in1 := "hours motors".MC_03_MIN, in2 := 60)
      { S7_GenerateENO := "TRUE" } Move(in := 1, out1 => "hours motors".MC_03_HOUR)
      { S7_GenerateENO := "TRUE" } Move(in := 0, out1 => "hours motors".MC_03_MIN)
      S_Coil( "Flag_Aggiorna_DB" )
   END_RUNG
   // the same network as SCL:
   // ENO of a box is taken as its EN; it also drops when the box reports an error
   #_w1 := "Tag_47" AND "102A7_SPARE5";
   IF #_w1 THEN "hours motors".MC_03_MIN := "hours motors".MC_03_MIN + 1; END_IF;
   IF #_w1 AND ("hours motors".MC_03_MIN >= 60) THEN "hours motors".MC_03_HOUR := 1; END_IF;
   #_w2 := #_w1 AND ("hours motors".MC_03_MIN >= 60);
   IF #_w2 THEN
       "hours motors".MC_03_MIN := 0;
       "Flag_Aggiorna_DB" := TRUE;
   END_IF;
END_REGION

REGION Network 21: MC-04
   RUNG wire#powerrail
      Contact( "Tag_47" )
      Contact( "MC04_Fbk" )
      wire#w1
      { S7_Templates := "SrcType := Int"; S7_GenerateENO := "TRUE" } Add(in1 := "hours motors".MC_04_MIN, in2 := 1, out => "hours motors".MC_04_MIN)
   END_RUNG
   RUNG wire#w1
      { S7_Templates := "SrcType := Int" } GE_Contact(in1 := "hours motors".MC_04_MIN, in2 := 60)
      { S7_GenerateENO := "TRUE" } Move(in := 1, out1 => "hours motors".MC_04_HOUR)
      { S7_GenerateENO := "TRUE" } Move(in := 0, out1 => "hours motors".MC_04_MIN)
      S_Coil( "Flag_Aggiorna_DB" )
   END_RUNG
   // the same network as SCL:
   // ENO of a box is taken as its EN; it also drops when the box reports an error
   #_w1 := "Tag_47" AND "MC04_Fbk";
   IF #_w1 THEN "hours motors".MC_04_MIN := "hours motors".MC_04_MIN + 1; END_IF;
   IF #_w1 AND ("hours motors".MC_04_MIN >= 60) THEN "hours motors".MC_04_HOUR := 1; END_IF;
   #_w2 := #_w1 AND ("hours motors".MC_04_MIN >= 60);
   IF #_w2 THEN
       "hours motors".MC_04_MIN := 0;
       "Flag_Aggiorna_DB" := TRUE;
   END_IF;
END_REGION

REGION Network 22: MC-05 / MC-05 DELETED
END_REGION

REGION Network 23: VS-01
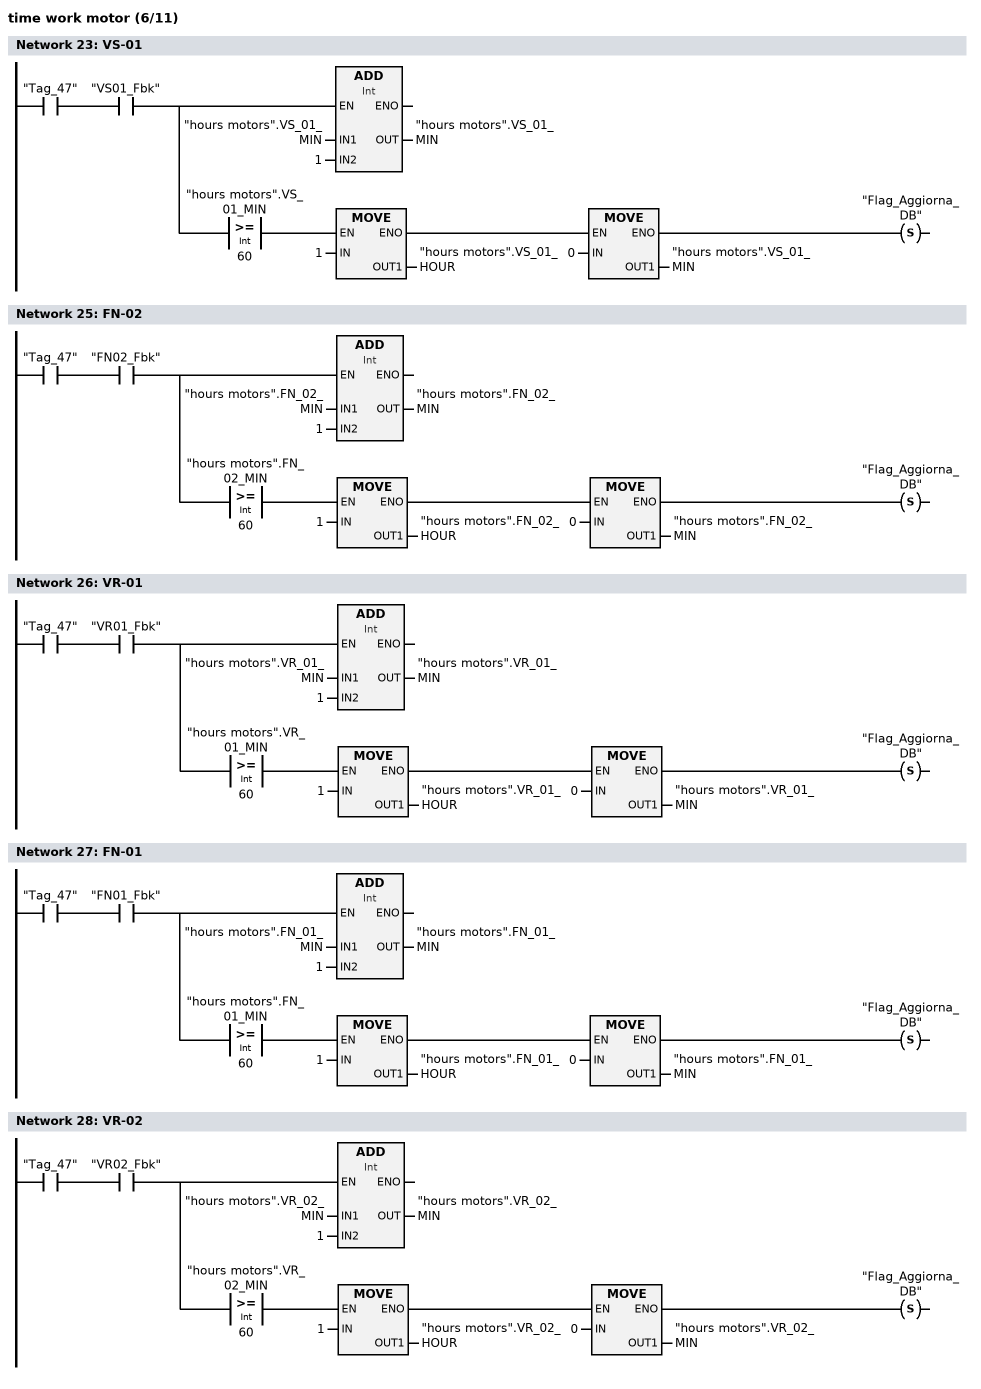
   RUNG wire#powerrail
      Contact( "Tag_47" )
      Contact( "VS01_Fbk" )
      wire#w1
      { S7_Templates := "SrcType := Int"; S7_GenerateENO := "TRUE" } Add(in1 := "hours motors".VS_01_MIN, in2 := 1, out => "hours motors".VS_01_MIN)
   END_RUNG
   RUNG wire#w1
      { S7_Templates := "SrcType := Int" } GE_Contact(in1 := "hours motors".VS_01_MIN, in2 := 60)
      { S7_GenerateENO := "TRUE" } Move(in := 1, out1 => "hours motors".VS_01_HOUR)
      { S7_GenerateENO := "TRUE" } Move(in := 0, out1 => "hours motors".VS_01_MIN)
      S_Coil( "Flag_Aggiorna_DB" )
   END_RUNG
   // the same network as SCL:
   // ENO of a box is taken as its EN; it also drops when the box reports an error
   #_w1 := "Tag_47" AND "VS01_Fbk";
   IF #_w1 THEN "hours motors".VS_01_MIN := "hours motors".VS_01_MIN + 1; END_IF;
   IF #_w1 AND ("hours motors".VS_01_MIN >= 60) THEN "hours motors".VS_01_HOUR := 1; END_IF;
   #_w2 := #_w1 AND ("hours motors".VS_01_MIN >= 60);
   IF #_w2 THEN
       "hours motors".VS_01_MIN := 0;
       "Flag_Aggiorna_DB" := TRUE;
   END_IF;
END_REGION

REGION Network 24: SC-12 / SC-12 DELETED
END_REGION

REGION Network 25: FN-02
   RUNG wire#powerrail
      Contact( "Tag_47" )
      Contact( "FN02_Fbk" )
      wire#w1
      { S7_Templates := "SrcType := Int"; S7_GenerateENO := "TRUE" } Add(in1 := "hours motors".FN_02_MIN, in2 := 1, out => "hours motors".FN_02_MIN)
   END_RUNG
   RUNG wire#w1
      { S7_Templates := "SrcType := Int" } GE_Contact(in1 := "hours motors".FN_02_MIN, in2 := 60)
      { S7_GenerateENO := "TRUE" } Move(in := 1, out1 => "hours motors".FN_02_HOUR)
      { S7_GenerateENO := "TRUE" } Move(in := 0, out1 => "hours motors".FN_02_MIN)
      S_Coil( "Flag_Aggiorna_DB" )
   END_RUNG
   // the same network as SCL:
   // ENO of a box is taken as its EN; it also drops when the box reports an error
   #_w1 := "Tag_47" AND "FN02_Fbk";
   IF #_w1 THEN "hours motors".FN_02_MIN := "hours motors".FN_02_MIN + 1; END_IF;
   IF #_w1 AND ("hours motors".FN_02_MIN >= 60) THEN "hours motors".FN_02_HOUR := 1; END_IF;
   #_w2 := #_w1 AND ("hours motors".FN_02_MIN >= 60);
   IF #_w2 THEN
       "hours motors".FN_02_MIN := 0;
       "Flag_Aggiorna_DB" := TRUE;
   END_IF;
END_REGION

REGION Network 26: VR-01
   RUNG wire#powerrail
      Contact( "Tag_47" )
      Contact( "VR01_Fbk" )
      wire#w1
      { S7_Templates := "SrcType := Int"; S7_GenerateENO := "TRUE" } Add(in1 := "hours motors".VR_01_MIN, in2 := 1, out => "hours motors".VR_01_MIN)
   END_RUNG
   RUNG wire#w1
      { S7_Templates := "SrcType := Int" } GE_Contact(in1 := "hours motors".VR_01_MIN, in2 := 60)
      { S7_GenerateENO := "TRUE" } Move(in := 1, out1 => "hours motors".VR_01_HOUR)
      { S7_GenerateENO := "TRUE" } Move(in := 0, out1 => "hours motors".VR_01_MIN)
      S_Coil( "Flag_Aggiorna_DB" )
   END_RUNG
   // the same network as SCL:
   // ENO of a box is taken as its EN; it also drops when the box reports an error
   #_w1 := "Tag_47" AND "VR01_Fbk";
   IF #_w1 THEN "hours motors".VR_01_MIN := "hours motors".VR_01_MIN + 1; END_IF;
   IF #_w1 AND ("hours motors".VR_01_MIN >= 60) THEN "hours motors".VR_01_HOUR := 1; END_IF;
   #_w2 := #_w1 AND ("hours motors".VR_01_MIN >= 60);
   IF #_w2 THEN
       "hours motors".VR_01_MIN := 0;
       "Flag_Aggiorna_DB" := TRUE;
   END_IF;
END_REGION

REGION Network 27: FN-01
   RUNG wire#powerrail
      Contact( "Tag_47" )
      Contact( "FN01_Fbk" )
      wire#w1
      { S7_Templates := "SrcType := Int"; S7_GenerateENO := "TRUE" } Add(in1 := "hours motors".FN_01_MIN, in2 := 1, out => "hours motors".FN_01_MIN)
   END_RUNG
   RUNG wire#w1
      { S7_Templates := "SrcType := Int" } GE_Contact(in1 := "hours motors".FN_01_MIN, in2 := 60)
      { S7_GenerateENO := "TRUE" } Move(in := 1, out1 => "hours motors".FN_01_HOUR)
      { S7_GenerateENO := "TRUE" } Move(in := 0, out1 => "hours motors".FN_01_MIN)
      S_Coil( "Flag_Aggiorna_DB" )
   END_RUNG
   // the same network as SCL:
   // ENO of a box is taken as its EN; it also drops when the box reports an error
   #_w1 := "Tag_47" AND "FN01_Fbk";
   IF #_w1 THEN "hours motors".FN_01_MIN := "hours motors".FN_01_MIN + 1; END_IF;
   IF #_w1 AND ("hours motors".FN_01_MIN >= 60) THEN "hours motors".FN_01_HOUR := 1; END_IF;
   #_w2 := #_w1 AND ("hours motors".FN_01_MIN >= 60);
   IF #_w2 THEN
       "hours motors".FN_01_MIN := 0;
       "Flag_Aggiorna_DB" := TRUE;
   END_IF;
END_REGION

REGION Network 28: VR-02
   RUNG wire#powerrail
      Contact( "Tag_47" )
      Contact( "VR02_Fbk" )
      wire#w1
      { S7_Templates := "SrcType := Int"; S7_GenerateENO := "TRUE" } Add(in1 := "hours motors".VR_02_MIN, in2 := 1, out => "hours motors".VR_02_MIN)
   END_RUNG
   RUNG wire#w1
      { S7_Templates := "SrcType := Int" } GE_Contact(in1 := "hours motors".VR_02_MIN, in2 := 60)
      { S7_GenerateENO := "TRUE" } Move(in := 1, out1 => "hours motors".VR_02_HOUR)
      { S7_GenerateENO := "TRUE" } Move(in := 0, out1 => "hours motors".VR_02_MIN)
      S_Coil( "Flag_Aggiorna_DB" )
   END_RUNG
   // the same network as SCL:
   // ENO of a box is taken as its EN; it also drops when the box reports an error
   #_w1 := "Tag_47" AND "VR02_Fbk";
   IF #_w1 THEN "hours motors".VR_02_MIN := "hours motors".VR_02_MIN + 1; END_IF;
   IF #_w1 AND ("hours motors".VR_02_MIN >= 60) THEN "hours motors".VR_02_HOUR := 1; END_IF;
   #_w2 := #_w1 AND ("hours motors".VR_02_MIN >= 60);
   IF #_w2 THEN
       "hours motors".VR_02_MIN := 0;
       "Flag_Aggiorna_DB" := TRUE;
   END_IF;
END_REGION

REGION Network 29: CH-01
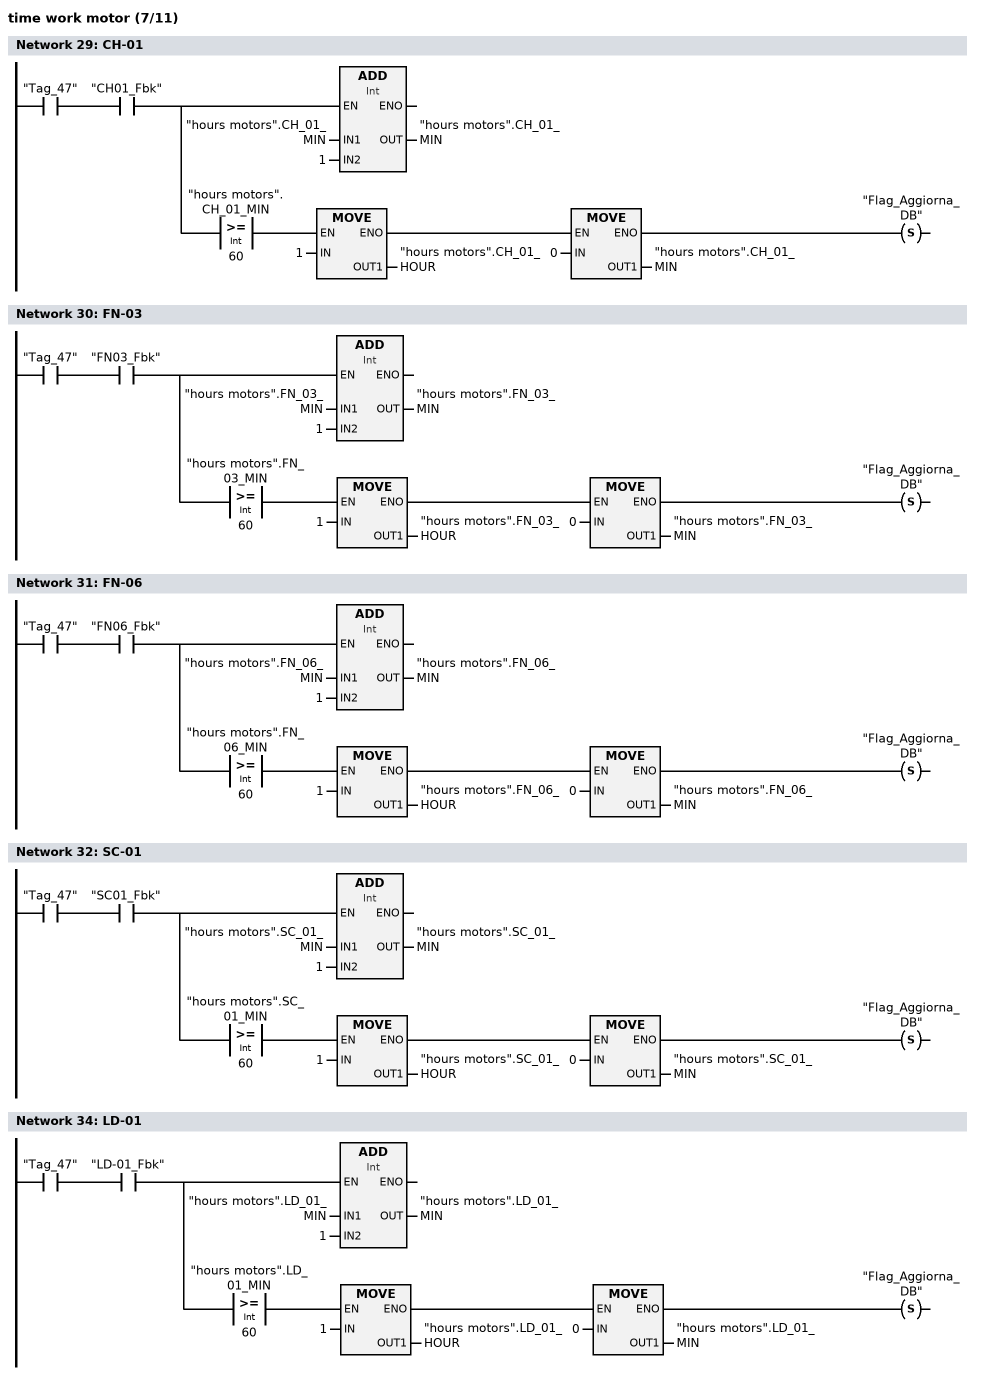
   RUNG wire#powerrail
      Contact( "Tag_47" )
      Contact( "CH01_Fbk" )
      wire#w1
      { S7_Templates := "SrcType := Int"; S7_GenerateENO := "TRUE" } Add(in1 := "hours motors".CH_01_MIN, in2 := 1, out => "hours motors".CH_01_MIN)
   END_RUNG
   RUNG wire#w1
      { S7_Templates := "SrcType := Int" } GE_Contact(in1 := "hours motors".CH_01_MIN, in2 := 60)
      { S7_GenerateENO := "TRUE" } Move(in := 1, out1 => "hours motors".CH_01_HOUR)
      { S7_GenerateENO := "TRUE" } Move(in := 0, out1 => "hours motors".CH_01_MIN)
      S_Coil( "Flag_Aggiorna_DB" )
   END_RUNG
   // the same network as SCL:
   // ENO of a box is taken as its EN; it also drops when the box reports an error
   #_w1 := "Tag_47" AND "CH01_Fbk";
   IF #_w1 THEN "hours motors".CH_01_MIN := "hours motors".CH_01_MIN + 1; END_IF;
   IF #_w1 AND ("hours motors".CH_01_MIN >= 60) THEN "hours motors".CH_01_HOUR := 1; END_IF;
   #_w2 := #_w1 AND ("hours motors".CH_01_MIN >= 60);
   IF #_w2 THEN
       "hours motors".CH_01_MIN := 0;
       "Flag_Aggiorna_DB" := TRUE;
   END_IF;
END_REGION

REGION Network 30: FN-03
   RUNG wire#powerrail
      Contact( "Tag_47" )
      Contact( "FN03_Fbk" )
      wire#w1
      { S7_Templates := "SrcType := Int"; S7_GenerateENO := "TRUE" } Add(in1 := "hours motors".FN_03_MIN, in2 := 1, out => "hours motors".FN_03_MIN)
   END_RUNG
   RUNG wire#w1
      { S7_Templates := "SrcType := Int" } GE_Contact(in1 := "hours motors".FN_03_MIN, in2 := 60)
      { S7_GenerateENO := "TRUE" } Move(in := 1, out1 => "hours motors".FN_03_HOUR)
      { S7_GenerateENO := "TRUE" } Move(in := 0, out1 => "hours motors".FN_03_MIN)
      S_Coil( "Flag_Aggiorna_DB" )
   END_RUNG
   // the same network as SCL:
   // ENO of a box is taken as its EN; it also drops when the box reports an error
   #_w1 := "Tag_47" AND "FN03_Fbk";
   IF #_w1 THEN "hours motors".FN_03_MIN := "hours motors".FN_03_MIN + 1; END_IF;
   IF #_w1 AND ("hours motors".FN_03_MIN >= 60) THEN "hours motors".FN_03_HOUR := 1; END_IF;
   #_w2 := #_w1 AND ("hours motors".FN_03_MIN >= 60);
   IF #_w2 THEN
       "hours motors".FN_03_MIN := 0;
       "Flag_Aggiorna_DB" := TRUE;
   END_IF;
END_REGION

REGION Network 31: FN-06
   RUNG wire#powerrail
      Contact( "Tag_47" )
      Contact( "FN06_Fbk" )
      wire#w1
      { S7_Templates := "SrcType := Int"; S7_GenerateENO := "TRUE" } Add(in1 := "hours motors".FN_06_MIN, in2 := 1, out => "hours motors".FN_06_MIN)
   END_RUNG
   RUNG wire#w1
      { S7_Templates := "SrcType := Int" } GE_Contact(in1 := "hours motors".FN_06_MIN, in2 := 60)
      { S7_GenerateENO := "TRUE" } Move(in := 1, out1 => "hours motors".FN_06_HOUR)
      { S7_GenerateENO := "TRUE" } Move(in := 0, out1 => "hours motors".FN_06_MIN)
      S_Coil( "Flag_Aggiorna_DB" )
   END_RUNG
   // the same network as SCL:
   // ENO of a box is taken as its EN; it also drops when the box reports an error
   #_w1 := "Tag_47" AND "FN06_Fbk";
   IF #_w1 THEN "hours motors".FN_06_MIN := "hours motors".FN_06_MIN + 1; END_IF;
   IF #_w1 AND ("hours motors".FN_06_MIN >= 60) THEN "hours motors".FN_06_HOUR := 1; END_IF;
   #_w2 := #_w1 AND ("hours motors".FN_06_MIN >= 60);
   IF #_w2 THEN
       "hours motors".FN_06_MIN := 0;
       "Flag_Aggiorna_DB" := TRUE;
   END_IF;
END_REGION

REGION Network 32: SC-01
   RUNG wire#powerrail
      Contact( "Tag_47" )
      Contact( "SC01_Fbk" )
      wire#w1
      { S7_Templates := "SrcType := Int"; S7_GenerateENO := "TRUE" } Add(in1 := "hours motors".SC_01_MIN, in2 := 1, out => "hours motors".SC_01_MIN)
   END_RUNG
   RUNG wire#w1
      { S7_Templates := "SrcType := Int" } GE_Contact(in1 := "hours motors".SC_01_MIN, in2 := 60)
      { S7_GenerateENO := "TRUE" } Move(in := 1, out1 => "hours motors".SC_01_HOUR)
      { S7_GenerateENO := "TRUE" } Move(in := 0, out1 => "hours motors".SC_01_MIN)
      S_Coil( "Flag_Aggiorna_DB" )
   END_RUNG
   // the same network as SCL:
   // ENO of a box is taken as its EN; it also drops when the box reports an error
   #_w1 := "Tag_47" AND "SC01_Fbk";
   IF #_w1 THEN "hours motors".SC_01_MIN := "hours motors".SC_01_MIN + 1; END_IF;
   IF #_w1 AND ("hours motors".SC_01_MIN >= 60) THEN "hours motors".SC_01_HOUR := 1; END_IF;
   #_w2 := #_w1 AND ("hours motors".SC_01_MIN >= 60);
   IF #_w2 THEN
       "hours motors".SC_01_MIN := 0;
       "Flag_Aggiorna_DB" := TRUE;
   END_IF;
END_REGION

REGION Network 33: FN-01 FAN / FN-01 FAN DELETED
END_REGION

REGION Network 34: LD-01
   RUNG wire#powerrail
      Contact( "Tag_47" )
      Contact( "LD-01_Fbk" )
      wire#w1
      { S7_Templates := "SrcType := Int"; S7_GenerateENO := "TRUE" } Add(in1 := "hours motors".LD_01_MIN, in2 := 1, out => "hours motors".LD_01_MIN)
   END_RUNG
   RUNG wire#w1
      { S7_Templates := "SrcType := Int" } GE_Contact(in1 := "hours motors".LD_01_MIN, in2 := 60)
      { S7_GenerateENO := "TRUE" } Move(in := 1, out1 => "hours motors".LD_01_HOUR)
      { S7_GenerateENO := "TRUE" } Move(in := 0, out1 => "hours motors".LD_01_MIN)
      S_Coil( "Flag_Aggiorna_DB" )
   END_RUNG
   // the same network as SCL:
   // ENO of a box is taken as its EN; it also drops when the box reports an error
   #_w1 := "Tag_47" AND "LD-01_Fbk";
   IF #_w1 THEN "hours motors".LD_01_MIN := "hours motors".LD_01_MIN + 1; END_IF;
   IF #_w1 AND ("hours motors".LD_01_MIN >= 60) THEN "hours motors".LD_01_HOUR := 1; END_IF;
   #_w2 := #_w1 AND ("hours motors".LD_01_MIN >= 60);
   IF #_w2 THEN
       "hours motors".LD_01_MIN := 0;
       "Flag_Aggiorna_DB" := TRUE;
   END_IF;
END_REGION

REGION Network 35: LD-01 VIB
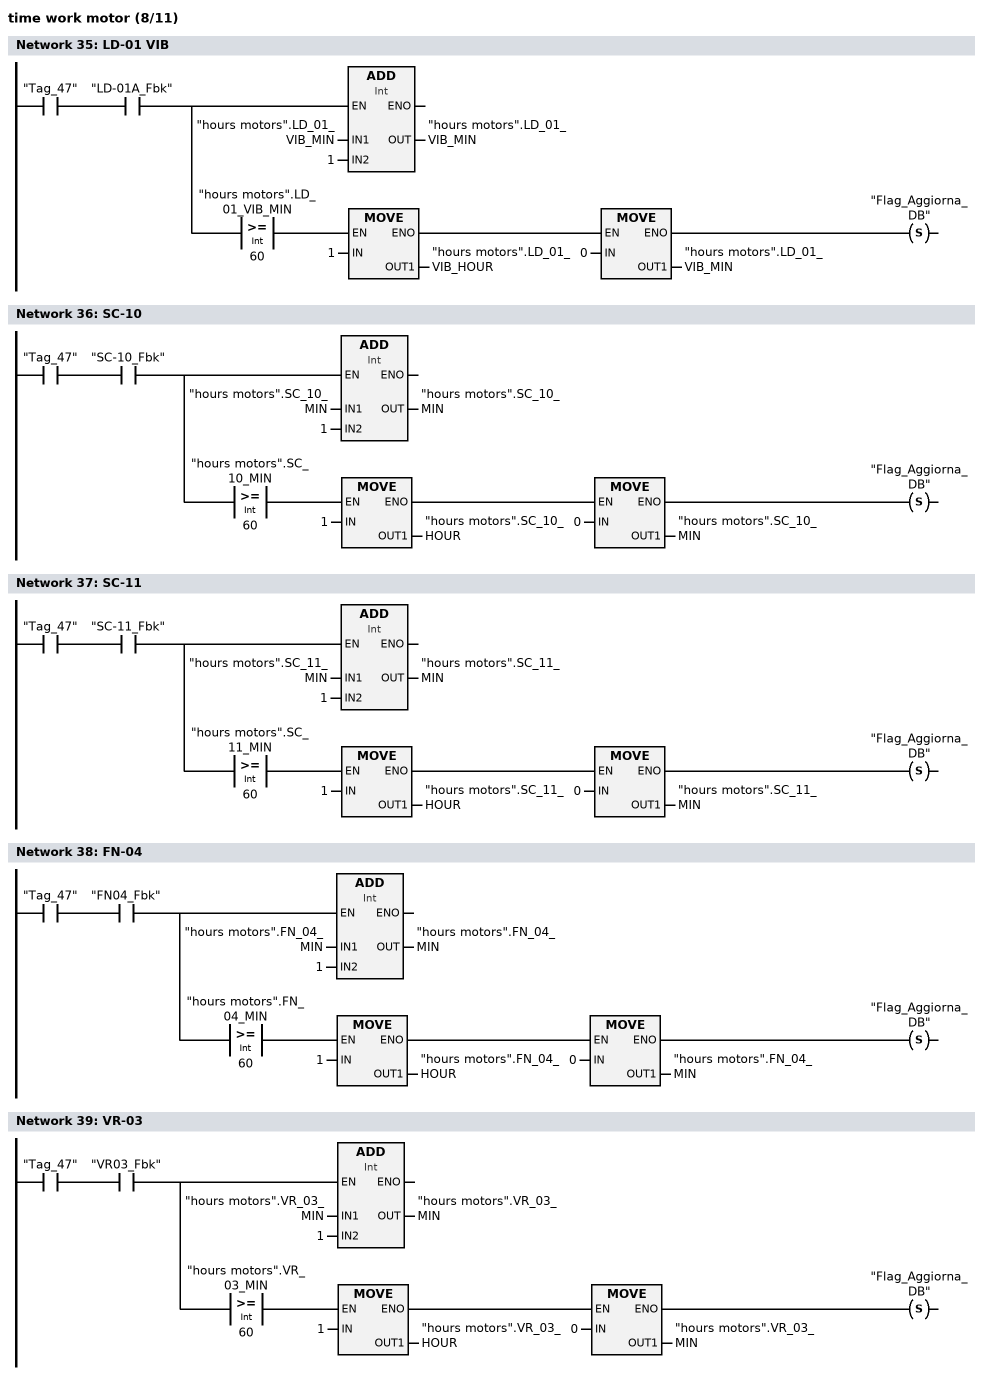
   RUNG wire#powerrail
      Contact( "Tag_47" )
      Contact( "LD-01A_Fbk" )
      wire#w1
      { S7_Templates := "SrcType := Int"; S7_GenerateENO := "TRUE" } Add(in1 := "hours motors".LD_01_VIB_MIN, in2 := 1, out => "hours motors".LD_01_VIB_MIN)
   END_RUNG
   RUNG wire#w1
      { S7_Templates := "SrcType := Int" } GE_Contact(in1 := "hours motors".LD_01_VIB_MIN, in2 := 60)
      { S7_GenerateENO := "TRUE" } Move(in := 1, out1 => "hours motors".LD_01_VIB_HOUR)
      { S7_GenerateENO := "TRUE" } Move(in := 0, out1 => "hours motors".LD_01_VIB_MIN)
      S_Coil( "Flag_Aggiorna_DB" )
   END_RUNG
   // the same network as SCL:
   // ENO of a box is taken as its EN; it also drops when the box reports an error
   #_w1 := "Tag_47" AND "LD-01A_Fbk";
   IF #_w1 THEN "hours motors".LD_01_VIB_MIN := "hours motors".LD_01_VIB_MIN + 1; END_IF;
   IF #_w1 AND ("hours motors".LD_01_VIB_MIN >= 60) THEN "hours motors".LD_01_VIB_HOUR := 1; END_IF;
   #_w2 := #_w1 AND ("hours motors".LD_01_VIB_MIN >= 60);
   IF #_w2 THEN
       "hours motors".LD_01_VIB_MIN := 0;
       "Flag_Aggiorna_DB" := TRUE;
   END_IF;
END_REGION

REGION Network 36: SC-10
   RUNG wire#powerrail
      Contact( "Tag_47" )
      Contact( "SC-10_Fbk" )
      wire#w1
      { S7_Templates := "SrcType := Int"; S7_GenerateENO := "TRUE" } Add(in1 := "hours motors".SC_10_MIN, in2 := 1, out => "hours motors".SC_10_MIN)
   END_RUNG
   RUNG wire#w1
      { S7_Templates := "SrcType := Int" } GE_Contact(in1 := "hours motors".SC_10_MIN, in2 := 60)
      { S7_GenerateENO := "TRUE" } Move(in := 1, out1 => "hours motors".SC_10_HOUR)
      { S7_GenerateENO := "TRUE" } Move(in := 0, out1 => "hours motors".SC_10_MIN)
      S_Coil( "Flag_Aggiorna_DB" )
   END_RUNG
   // the same network as SCL:
   // ENO of a box is taken as its EN; it also drops when the box reports an error
   #_w1 := "Tag_47" AND "SC-10_Fbk";
   IF #_w1 THEN "hours motors".SC_10_MIN := "hours motors".SC_10_MIN + 1; END_IF;
   IF #_w1 AND ("hours motors".SC_10_MIN >= 60) THEN "hours motors".SC_10_HOUR := 1; END_IF;
   #_w2 := #_w1 AND ("hours motors".SC_10_MIN >= 60);
   IF #_w2 THEN
       "hours motors".SC_10_MIN := 0;
       "Flag_Aggiorna_DB" := TRUE;
   END_IF;
END_REGION

REGION Network 37: SC-11
   RUNG wire#powerrail
      Contact( "Tag_47" )
      Contact( "SC-11_Fbk" )
      wire#w1
      { S7_Templates := "SrcType := Int"; S7_GenerateENO := "TRUE" } Add(in1 := "hours motors".SC_11_MIN, in2 := 1, out => "hours motors".SC_11_MIN)
   END_RUNG
   RUNG wire#w1
      { S7_Templates := "SrcType := Int" } GE_Contact(in1 := "hours motors".SC_11_MIN, in2 := 60)
      { S7_GenerateENO := "TRUE" } Move(in := 1, out1 => "hours motors".SC_11_HOUR)
      { S7_GenerateENO := "TRUE" } Move(in := 0, out1 => "hours motors".SC_11_MIN)
      S_Coil( "Flag_Aggiorna_DB" )
   END_RUNG
   // the same network as SCL:
   // ENO of a box is taken as its EN; it also drops when the box reports an error
   #_w1 := "Tag_47" AND "SC-11_Fbk";
   IF #_w1 THEN "hours motors".SC_11_MIN := "hours motors".SC_11_MIN + 1; END_IF;
   IF #_w1 AND ("hours motors".SC_11_MIN >= 60) THEN "hours motors".SC_11_HOUR := 1; END_IF;
   #_w2 := #_w1 AND ("hours motors".SC_11_MIN >= 60);
   IF #_w2 THEN
       "hours motors".SC_11_MIN := 0;
       "Flag_Aggiorna_DB" := TRUE;
   END_IF;
END_REGION

REGION Network 38: FN-04
   RUNG wire#powerrail
      Contact( "Tag_47" )
      Contact( "FN04_Fbk" )
      wire#w1
      { S7_Templates := "SrcType := Int"; S7_GenerateENO := "TRUE" } Add(in1 := "hours motors".FN_04_MIN, in2 := 1, out => "hours motors".FN_04_MIN)
   END_RUNG
   RUNG wire#w1
      { S7_Templates := "SrcType := Int" } GE_Contact(in1 := "hours motors".FN_04_MIN, in2 := 60)
      { S7_GenerateENO := "TRUE" } Move(in := 1, out1 => "hours motors".FN_04_HOUR)
      { S7_GenerateENO := "TRUE" } Move(in := 0, out1 => "hours motors".FN_04_MIN)
      S_Coil( "Flag_Aggiorna_DB" )
   END_RUNG
   // the same network as SCL:
   // ENO of a box is taken as its EN; it also drops when the box reports an error
   #_w1 := "Tag_47" AND "FN04_Fbk";
   IF #_w1 THEN "hours motors".FN_04_MIN := "hours motors".FN_04_MIN + 1; END_IF;
   IF #_w1 AND ("hours motors".FN_04_MIN >= 60) THEN "hours motors".FN_04_HOUR := 1; END_IF;
   #_w2 := #_w1 AND ("hours motors".FN_04_MIN >= 60);
   IF #_w2 THEN
       "hours motors".FN_04_MIN := 0;
       "Flag_Aggiorna_DB" := TRUE;
   END_IF;
END_REGION

REGION Network 39: VR-03
   RUNG wire#powerrail
      Contact( "Tag_47" )
      Contact( "VR03_Fbk" )
      wire#w1
      { S7_Templates := "SrcType := Int"; S7_GenerateENO := "TRUE" } Add(in1 := "hours motors".VR_03_MIN, in2 := 1, out => "hours motors".VR_03_MIN)
   END_RUNG
   RUNG wire#w1
      { S7_Templates := "SrcType := Int" } GE_Contact(in1 := "hours motors".VR_03_MIN, in2 := 60)
      { S7_GenerateENO := "TRUE" } Move(in := 1, out1 => "hours motors".VR_03_HOUR)
      { S7_GenerateENO := "TRUE" } Move(in := 0, out1 => "hours motors".VR_03_MIN)
      S_Coil( "Flag_Aggiorna_DB" )
   END_RUNG
   // the same network as SCL:
   // ENO of a box is taken as its EN; it also drops when the box reports an error
   #_w1 := "Tag_47" AND "VR03_Fbk";
   IF #_w1 THEN "hours motors".VR_03_MIN := "hours motors".VR_03_MIN + 1; END_IF;
   IF #_w1 AND ("hours motors".VR_03_MIN >= 60) THEN "hours motors".VR_03_HOUR := 1; END_IF;
   #_w2 := #_w1 AND ("hours motors".VR_03_MIN >= 60);
   IF #_w2 THEN
       "hours motors".VR_03_MIN := 0;
       "Flag_Aggiorna_DB" := TRUE;
   END_IF;
END_REGION

REGION Network 40: VR-04
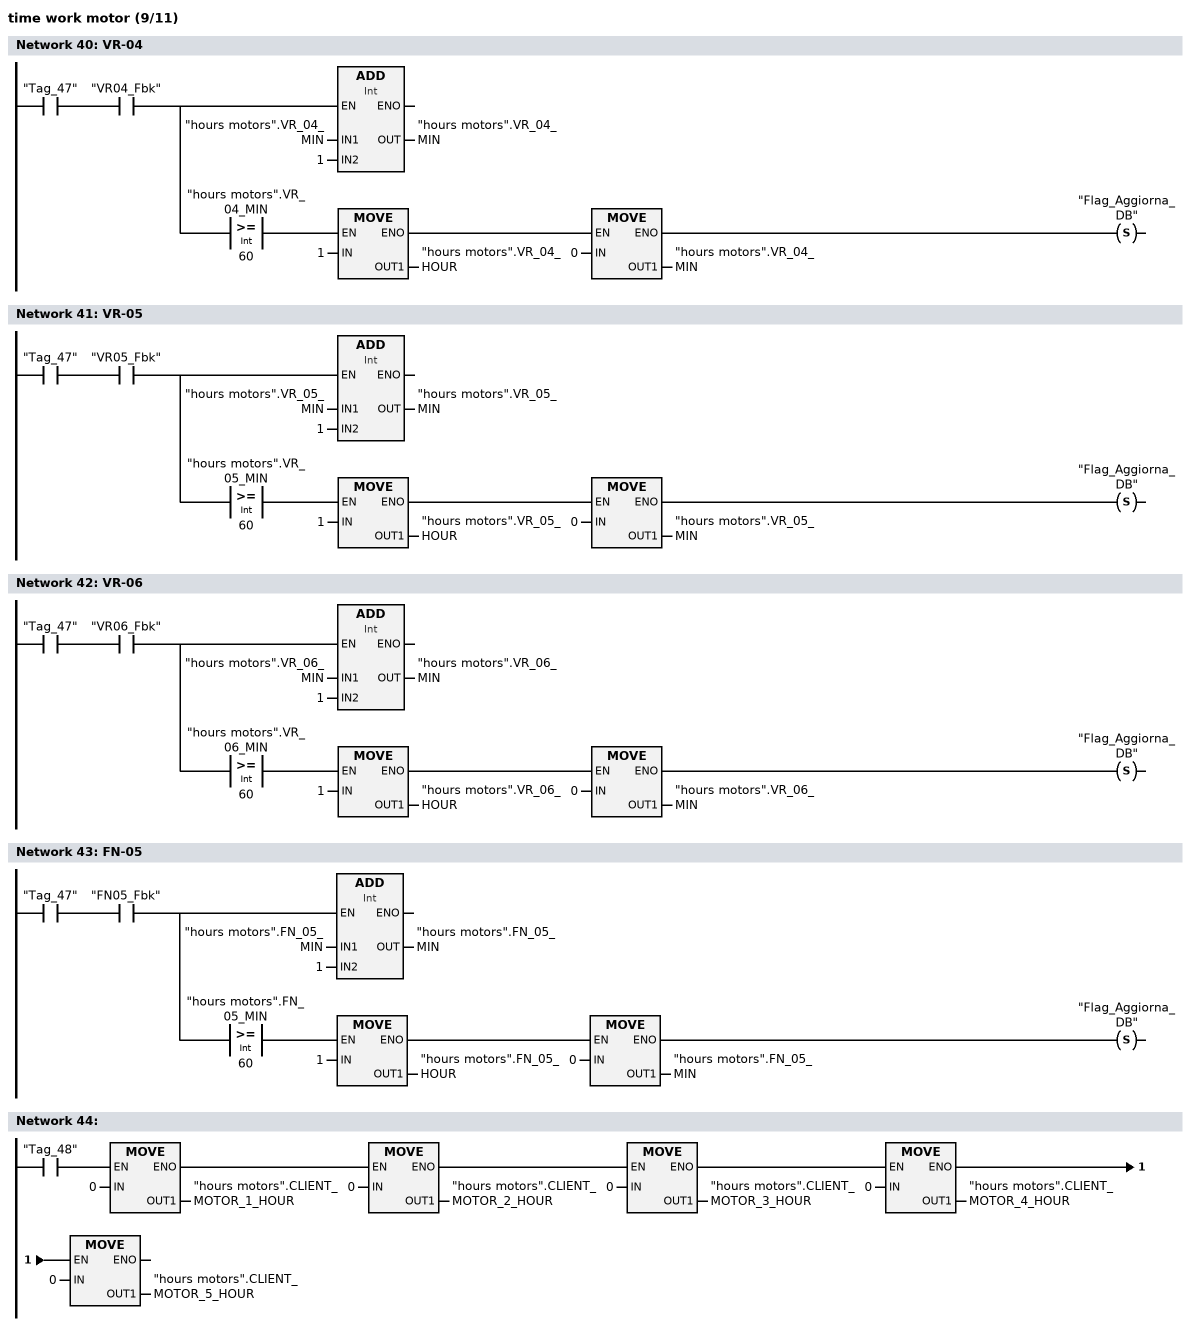
   RUNG wire#powerrail
      Contact( "Tag_47" )
      Contact( "VR04_Fbk" )
      wire#w1
      { S7_Templates := "SrcType := Int"; S7_GenerateENO := "TRUE" } Add(in1 := "hours motors".VR_04_MIN, in2 := 1, out => "hours motors".VR_04_MIN)
   END_RUNG
   RUNG wire#w1
      { S7_Templates := "SrcType := Int" } GE_Contact(in1 := "hours motors".VR_04_MIN, in2 := 60)
      { S7_GenerateENO := "TRUE" } Move(in := 1, out1 => "hours motors".VR_04_HOUR)
      { S7_GenerateENO := "TRUE" } Move(in := 0, out1 => "hours motors".VR_04_MIN)
      S_Coil( "Flag_Aggiorna_DB" )
   END_RUNG
   // the same network as SCL:
   // ENO of a box is taken as its EN; it also drops when the box reports an error
   #_w1 := "Tag_47" AND "VR04_Fbk";
   IF #_w1 THEN "hours motors".VR_04_MIN := "hours motors".VR_04_MIN + 1; END_IF;
   IF #_w1 AND ("hours motors".VR_04_MIN >= 60) THEN "hours motors".VR_04_HOUR := 1; END_IF;
   #_w2 := #_w1 AND ("hours motors".VR_04_MIN >= 60);
   IF #_w2 THEN
       "hours motors".VR_04_MIN := 0;
       "Flag_Aggiorna_DB" := TRUE;
   END_IF;
END_REGION

REGION Network 41: VR-05
   RUNG wire#powerrail
      Contact( "Tag_47" )
      Contact( "VR05_Fbk" )
      wire#w1
      { S7_Templates := "SrcType := Int"; S7_GenerateENO := "TRUE" } Add(in1 := "hours motors".VR_05_MIN, in2 := 1, out => "hours motors".VR_05_MIN)
   END_RUNG
   RUNG wire#w1
      { S7_Templates := "SrcType := Int" } GE_Contact(in1 := "hours motors".VR_05_MIN, in2 := 60)
      { S7_GenerateENO := "TRUE" } Move(in := 1, out1 => "hours motors".VR_05_HOUR)
      { S7_GenerateENO := "TRUE" } Move(in := 0, out1 => "hours motors".VR_05_MIN)
      S_Coil( "Flag_Aggiorna_DB" )
   END_RUNG
   // the same network as SCL:
   // ENO of a box is taken as its EN; it also drops when the box reports an error
   #_w1 := "Tag_47" AND "VR05_Fbk";
   IF #_w1 THEN "hours motors".VR_05_MIN := "hours motors".VR_05_MIN + 1; END_IF;
   IF #_w1 AND ("hours motors".VR_05_MIN >= 60) THEN "hours motors".VR_05_HOUR := 1; END_IF;
   #_w2 := #_w1 AND ("hours motors".VR_05_MIN >= 60);
   IF #_w2 THEN
       "hours motors".VR_05_MIN := 0;
       "Flag_Aggiorna_DB" := TRUE;
   END_IF;
END_REGION

REGION Network 42: VR-06
   RUNG wire#powerrail
      Contact( "Tag_47" )
      Contact( "VR06_Fbk" )
      wire#w1
      { S7_Templates := "SrcType := Int"; S7_GenerateENO := "TRUE" } Add(in1 := "hours motors".VR_06_MIN, in2 := 1, out => "hours motors".VR_06_MIN)
   END_RUNG
   RUNG wire#w1
      { S7_Templates := "SrcType := Int" } GE_Contact(in1 := "hours motors".VR_06_MIN, in2 := 60)
      { S7_GenerateENO := "TRUE" } Move(in := 1, out1 => "hours motors".VR_06_HOUR)
      { S7_GenerateENO := "TRUE" } Move(in := 0, out1 => "hours motors".VR_06_MIN)
      S_Coil( "Flag_Aggiorna_DB" )
   END_RUNG
   // the same network as SCL:
   // ENO of a box is taken as its EN; it also drops when the box reports an error
   #_w1 := "Tag_47" AND "VR06_Fbk";
   IF #_w1 THEN "hours motors".VR_06_MIN := "hours motors".VR_06_MIN + 1; END_IF;
   IF #_w1 AND ("hours motors".VR_06_MIN >= 60) THEN "hours motors".VR_06_HOUR := 1; END_IF;
   #_w2 := #_w1 AND ("hours motors".VR_06_MIN >= 60);
   IF #_w2 THEN
       "hours motors".VR_06_MIN := 0;
       "Flag_Aggiorna_DB" := TRUE;
   END_IF;
END_REGION

REGION Network 43: FN-05
   RUNG wire#powerrail
      Contact( "Tag_47" )
      Contact( "FN05_Fbk" )
      wire#w1
      { S7_Templates := "SrcType := Int"; S7_GenerateENO := "TRUE" } Add(in1 := "hours motors".FN_05_MIN, in2 := 1, out => "hours motors".FN_05_MIN)
   END_RUNG
   RUNG wire#w1
      { S7_Templates := "SrcType := Int" } GE_Contact(in1 := "hours motors".FN_05_MIN, in2 := 60)
      { S7_GenerateENO := "TRUE" } Move(in := 1, out1 => "hours motors".FN_05_HOUR)
      { S7_GenerateENO := "TRUE" } Move(in := 0, out1 => "hours motors".FN_05_MIN)
      S_Coil( "Flag_Aggiorna_DB" )
   END_RUNG
   // the same network as SCL:
   // ENO of a box is taken as its EN; it also drops when the box reports an error
   #_w1 := "Tag_47" AND "FN05_Fbk";
   IF #_w1 THEN "hours motors".FN_05_MIN := "hours motors".FN_05_MIN + 1; END_IF;
   IF #_w1 AND ("hours motors".FN_05_MIN >= 60) THEN "hours motors".FN_05_HOUR := 1; END_IF;
   #_w2 := #_w1 AND ("hours motors".FN_05_MIN >= 60);
   IF #_w2 THEN
       "hours motors".FN_05_MIN := 0;
       "Flag_Aggiorna_DB" := TRUE;
   END_IF;
END_REGION

REGION Network 44
   RUNG wire#powerrail
      Contact( "Tag_48" )
      { S7_GenerateENO := "TRUE" } Move(in := 0, out1 => "hours motors".CLIENT_MOTOR_1_HOUR)
      { S7_GenerateENO := "TRUE" } Move(in := 0, out1 => "hours motors".CLIENT_MOTOR_2_HOUR)
      { S7_GenerateENO := "TRUE" } Move(in := 0, out1 => "hours motors".CLIENT_MOTOR_3_HOUR)
      { S7_GenerateENO := "TRUE" } Move(in := 0, out1 => "hours motors".CLIENT_MOTOR_4_HOUR)
      { S7_GenerateENO := "TRUE" } Move(in := 0, out1 => "hours motors".CLIENT_MOTOR_5_HOUR)
   END_RUNG
   // the same network as SCL:
   // ENO of a box is taken as its EN; it also drops when the box reports an error
   IF "Tag_48" THEN
       "hours motors".CLIENT_MOTOR_1_HOUR := 0;
       "hours motors".CLIENT_MOTOR_2_HOUR := 0;
       "hours motors".CLIENT_MOTOR_3_HOUR := 0;
       "hours motors".CLIENT_MOTOR_4_HOUR := 0;
       "hours motors".CLIENT_MOTOR_5_HOUR := 0;
   END_IF;
END_REGION

REGION Network 45
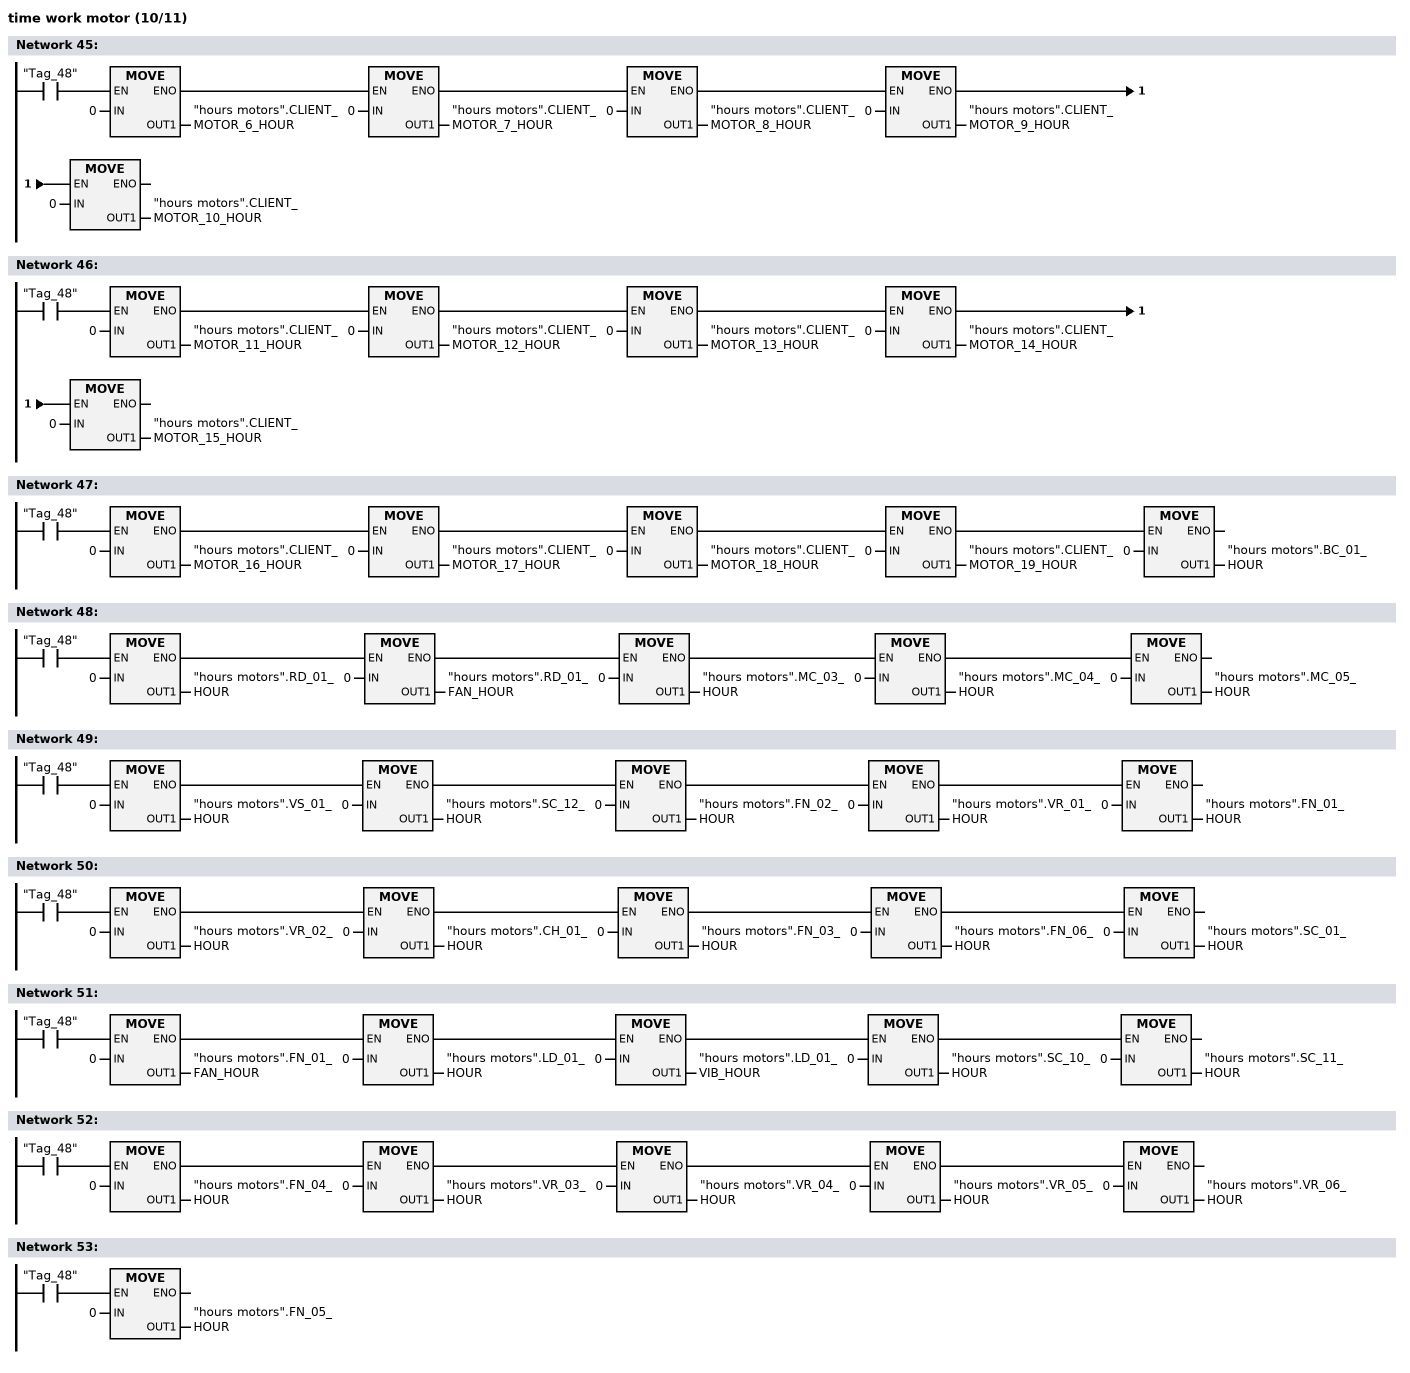
   RUNG wire#powerrail
      Contact( "Tag_48" )
      { S7_GenerateENO := "TRUE" } Move(in := 0, out1 => "hours motors".CLIENT_MOTOR_6_HOUR)
      { S7_GenerateENO := "TRUE" } Move(in := 0, out1 => "hours motors".CLIENT_MOTOR_7_HOUR)
      { S7_GenerateENO := "TRUE" } Move(in := 0, out1 => "hours motors".CLIENT_MOTOR_8_HOUR)
      { S7_GenerateENO := "TRUE" } Move(in := 0, out1 => "hours motors".CLIENT_MOTOR_9_HOUR)
      { S7_GenerateENO := "TRUE" } Move(in := 0, out1 => "hours motors".CLIENT_MOTOR_10_HOUR)
   END_RUNG
   // the same network as SCL:
   // ENO of a box is taken as its EN; it also drops when the box reports an error
   IF "Tag_48" THEN
       "hours motors".CLIENT_MOTOR_6_HOUR := 0;
       "hours motors".CLIENT_MOTOR_7_HOUR := 0;
       "hours motors".CLIENT_MOTOR_8_HOUR := 0;
       "hours motors".CLIENT_MOTOR_9_HOUR := 0;
       "hours motors".CLIENT_MOTOR_10_HOUR := 0;
   END_IF;
END_REGION

REGION Network 46
   RUNG wire#powerrail
      Contact( "Tag_48" )
      { S7_GenerateENO := "TRUE" } Move(in := 0, out1 => "hours motors".CLIENT_MOTOR_11_HOUR)
      { S7_GenerateENO := "TRUE" } Move(in := 0, out1 => "hours motors".CLIENT_MOTOR_12_HOUR)
      { S7_GenerateENO := "TRUE" } Move(in := 0, out1 => "hours motors".CLIENT_MOTOR_13_HOUR)
      { S7_GenerateENO := "TRUE" } Move(in := 0, out1 => "hours motors".CLIENT_MOTOR_14_HOUR)
      { S7_GenerateENO := "TRUE" } Move(in := 0, out1 => "hours motors".CLIENT_MOTOR_15_HOUR)
   END_RUNG
   // the same network as SCL:
   // ENO of a box is taken as its EN; it also drops when the box reports an error
   IF "Tag_48" THEN
       "hours motors".CLIENT_MOTOR_11_HOUR := 0;
       "hours motors".CLIENT_MOTOR_12_HOUR := 0;
       "hours motors".CLIENT_MOTOR_13_HOUR := 0;
       "hours motors".CLIENT_MOTOR_14_HOUR := 0;
       "hours motors".CLIENT_MOTOR_15_HOUR := 0;
   END_IF;
END_REGION

REGION Network 47
   RUNG wire#powerrail
      Contact( "Tag_48" )
      { S7_GenerateENO := "TRUE" } Move(in := 0, out1 => "hours motors".CLIENT_MOTOR_16_HOUR)
      { S7_GenerateENO := "TRUE" } Move(in := 0, out1 => "hours motors".CLIENT_MOTOR_17_HOUR)
      { S7_GenerateENO := "TRUE" } Move(in := 0, out1 => "hours motors".CLIENT_MOTOR_18_HOUR)
      { S7_GenerateENO := "TRUE" } Move(in := 0, out1 => "hours motors".CLIENT_MOTOR_19_HOUR)
      { S7_GenerateENO := "TRUE" } Move(in := 0, out1 => "hours motors".BC_01_HOUR)
   END_RUNG
   // the same network as SCL:
   // ENO of a box is taken as its EN; it also drops when the box reports an error
   IF "Tag_48" THEN
       "hours motors".CLIENT_MOTOR_16_HOUR := 0;
       "hours motors".CLIENT_MOTOR_17_HOUR := 0;
       "hours motors".CLIENT_MOTOR_18_HOUR := 0;
       "hours motors".CLIENT_MOTOR_19_HOUR := 0;
       "hours motors".BC_01_HOUR := 0;
   END_IF;
END_REGION

REGION Network 48
   RUNG wire#powerrail
      Contact( "Tag_48" )
      { S7_GenerateENO := "TRUE" } Move(in := 0, out1 => "hours motors".RD_01_HOUR)
      { S7_GenerateENO := "TRUE" } Move(in := 0, out1 => "hours motors".RD_01_FAN_HOUR)
      { S7_GenerateENO := "TRUE" } Move(in := 0, out1 => "hours motors".MC_03_HOUR)
      { S7_GenerateENO := "TRUE" } Move(in := 0, out1 => "hours motors".MC_04_HOUR)
      { S7_GenerateENO := "TRUE" } Move(in := 0, out1 => "hours motors".MC_05_HOUR)
   END_RUNG
   // the same network as SCL:
   // ENO of a box is taken as its EN; it also drops when the box reports an error
   IF "Tag_48" THEN
       "hours motors".RD_01_HOUR := 0;
       "hours motors".RD_01_FAN_HOUR := 0;
       "hours motors".MC_03_HOUR := 0;
       "hours motors".MC_04_HOUR := 0;
       "hours motors".MC_05_HOUR := 0;
   END_IF;
END_REGION

REGION Network 49
   RUNG wire#powerrail
      Contact( "Tag_48" )
      { S7_GenerateENO := "TRUE" } Move(in := 0, out1 => "hours motors".VS_01_HOUR)
      { S7_GenerateENO := "TRUE" } Move(in := 0, out1 => "hours motors".SC_12_HOUR)
      { S7_GenerateENO := "TRUE" } Move(in := 0, out1 => "hours motors".FN_02_HOUR)
      { S7_GenerateENO := "TRUE" } Move(in := 0, out1 => "hours motors".VR_01_HOUR)
      { S7_GenerateENO := "TRUE" } Move(in := 0, out1 => "hours motors".FN_01_HOUR)
   END_RUNG
   // the same network as SCL:
   // ENO of a box is taken as its EN; it also drops when the box reports an error
   IF "Tag_48" THEN
       "hours motors".VS_01_HOUR := 0;
       "hours motors".SC_12_HOUR := 0;
       "hours motors".FN_02_HOUR := 0;
       "hours motors".VR_01_HOUR := 0;
       "hours motors".FN_01_HOUR := 0;
   END_IF;
END_REGION

REGION Network 50
   RUNG wire#powerrail
      Contact( "Tag_48" )
      { S7_GenerateENO := "TRUE" } Move(in := 0, out1 => "hours motors".VR_02_HOUR)
      { S7_GenerateENO := "TRUE" } Move(in := 0, out1 => "hours motors".CH_01_HOUR)
      { S7_GenerateENO := "TRUE" } Move(in := 0, out1 => "hours motors".FN_03_HOUR)
      { S7_GenerateENO := "TRUE" } Move(in := 0, out1 => "hours motors".FN_06_HOUR)
      { S7_GenerateENO := "TRUE" } Move(in := 0, out1 => "hours motors".SC_01_HOUR)
   END_RUNG
   // the same network as SCL:
   // ENO of a box is taken as its EN; it also drops when the box reports an error
   IF "Tag_48" THEN
       "hours motors".VR_02_HOUR := 0;
       "hours motors".CH_01_HOUR := 0;
       "hours motors".FN_03_HOUR := 0;
       "hours motors".FN_06_HOUR := 0;
       "hours motors".SC_01_HOUR := 0;
   END_IF;
END_REGION

REGION Network 51
   RUNG wire#powerrail
      Contact( "Tag_48" )
      { S7_GenerateENO := "TRUE" } Move(in := 0, out1 => "hours motors".FN_01_FAN_HOUR)
      { S7_GenerateENO := "TRUE" } Move(in := 0, out1 => "hours motors".LD_01_HOUR)
      { S7_GenerateENO := "TRUE" } Move(in := 0, out1 => "hours motors".LD_01_VIB_HOUR)
      { S7_GenerateENO := "TRUE" } Move(in := 0, out1 => "hours motors".SC_10_HOUR)
      { S7_GenerateENO := "TRUE" } Move(in := 0, out1 => "hours motors".SC_11_HOUR)
   END_RUNG
   // the same network as SCL:
   // ENO of a box is taken as its EN; it also drops when the box reports an error
   IF "Tag_48" THEN
       "hours motors".FN_01_FAN_HOUR := 0;
       "hours motors".LD_01_HOUR := 0;
       "hours motors".LD_01_VIB_HOUR := 0;
       "hours motors".SC_10_HOUR := 0;
       "hours motors".SC_11_HOUR := 0;
   END_IF;
END_REGION

REGION Network 52
   RUNG wire#powerrail
      Contact( "Tag_48" )
      { S7_GenerateENO := "TRUE" } Move(in := 0, out1 => "hours motors".FN_04_HOUR)
      { S7_GenerateENO := "TRUE" } Move(in := 0, out1 => "hours motors".VR_03_HOUR)
      { S7_GenerateENO := "TRUE" } Move(in := 0, out1 => "hours motors".VR_04_HOUR)
      { S7_GenerateENO := "TRUE" } Move(in := 0, out1 => "hours motors".VR_05_HOUR)
      { S7_GenerateENO := "TRUE" } Move(in := 0, out1 => "hours motors".VR_06_HOUR)
   END_RUNG
   // the same network as SCL:
   // ENO of a box is taken as its EN; it also drops when the box reports an error
   IF "Tag_48" THEN
       "hours motors".FN_04_HOUR := 0;
       "hours motors".VR_03_HOUR := 0;
       "hours motors".VR_04_HOUR := 0;
       "hours motors".VR_05_HOUR := 0;
       "hours motors".VR_06_HOUR := 0;
   END_IF;
END_REGION

REGION Network 53
   RUNG wire#powerrail
      Contact( "Tag_48" )
      { S7_GenerateENO := "TRUE" } Move(in := 0, out1 => "hours motors".FN_05_HOUR)
   END_RUNG
   // the same network as SCL:
   IF "Tag_48" THEN "hours motors".FN_05_HOUR := 0; END_IF;
END_REGION

REGION Network 54: Reset ore di lavoro dopo che ha registrsato i dati nel DB / Reset working hours after recording the data in the DB
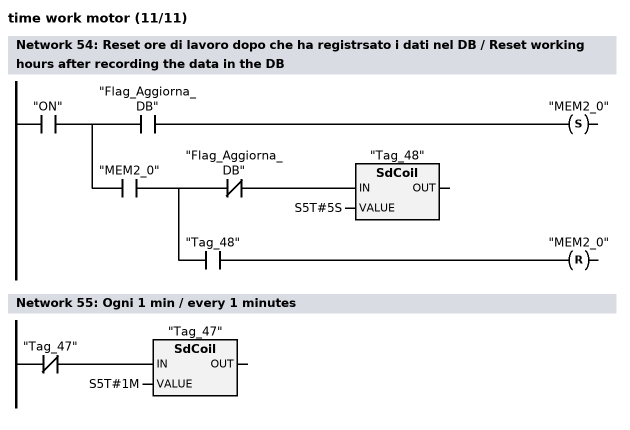
   // no SCL statement known for SdCoil: written as a call
   IF "ON" AND "Flag_Aggiorna_DB" THEN "MEM2_0" := TRUE; END_IF;
   #_w1 := "ON" AND "MEM2_0";
   SdCoil(in := #_w1 AND NOT "Flag_Aggiorna_DB", value := S5T#5S, operand := "Tag_48");
   IF #_w1 AND "Tag_48" THEN "MEM2_0" := FALSE; END_IF;
END_REGION

REGION Network 55: Ogni 1 min / every 1 minutes
   // no SCL statement known for SdCoil: written as a call
   SdCoil(in := NOT "Tag_47", value := S5T#1M, operand := "Tag_47");
END_REGION
END_FUNCTION

FUNCTION "Analog input conversion" : Void   // FC3, LAD
{ S7_Optimized_Access := 'FALSE' }
VERSION : 0.1
   VAR_TEMP
      TEMP0 : Int;
      TEMP1 : Int;
      TEMP2 : Int;
      Temp3 : Int;
      temp4 : Int;
      temp5 : Int;
      temp6 : Int;
      CNTV0_100 : DInt;
      CNTV1_100 : DInt;
      CNTV2_100 : DInt;
      CNTV3_100 : DInt;
      CNTV4_100 : DInt;
      CNTV5_100 : DInt;
      CNTV6_100 : DInt;
      CNTV7_100 : DInt;
      CNTV8_100 : DInt;
      CNT_Act_0 : DInt;
      CNT_Act_1 : DInt;
      CNT_Act_2 : DInt;
      CNT_Act_3 : DInt;
      CNT_Act_4 : DInt;
      temp7 : Int;
      JOB_NUMBER : Int;
   END_VAR
   VAR_TEMP   // added for the SCL form of the ladder/FBD networks
      _w1 : Bool;
      _w2 : Bool;
      _w3 : Bool;
      _w4 : Bool;
   END_VAR
BEGIN

REGION Network 1: TC04
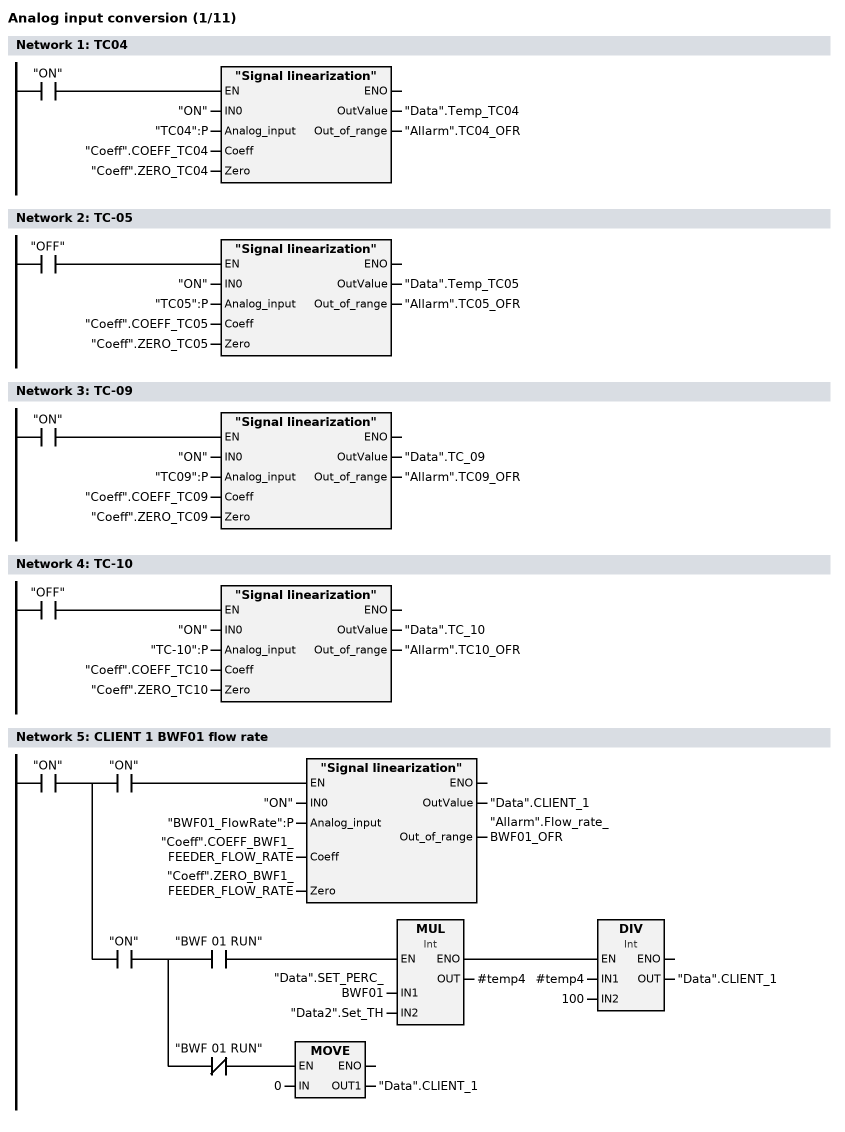
   RUNG wire#powerrail
      Contact( "ON" )
      "Signal linearization"(IN0 := "ON", Analog_input := "TC04":P, Coeff := "Coeff".COEFF_TC04, Zero := "Coeff".ZERO_TC04, OutValue => "Data".Temp_TC04, Out_of_range => "Allarm".TC04_OFR)
   END_RUNG
   // the same network as SCL:
   IF "ON" THEN
       "Signal linearization"(IN0 := "ON",
                              Analog_input := "TC04":P,
                              Coeff := "Coeff".COEFF_TC04,
                              Zero := "Coeff".ZERO_TC04,
                              OutValue => "Data".Temp_TC04,
                              Out_of_range => "Allarm".TC04_OFR);
   END_IF;
END_REGION

REGION Network 2: TC-05
   RUNG wire#powerrail
      Contact( "OFF" )
      "Signal linearization"(IN0 := "ON", Analog_input := "TC05":P, Coeff := "Coeff".COEFF_TC05, Zero := "Coeff".ZERO_TC05, OutValue => "Data".Temp_TC05, Out_of_range => "Allarm".TC05_OFR)
   END_RUNG
   // the same network as SCL:
   IF "OFF" THEN
       "Signal linearization"(IN0 := "ON",
                              Analog_input := "TC05":P,
                              Coeff := "Coeff".COEFF_TC05,
                              Zero := "Coeff".ZERO_TC05,
                              OutValue => "Data".Temp_TC05,
                              Out_of_range => "Allarm".TC05_OFR);
   END_IF;
END_REGION

REGION Network 3: TC-09
   RUNG wire#powerrail
      Contact( "ON" )
      "Signal linearization"(IN0 := "ON", Analog_input := "TC09":P, Coeff := "Coeff".COEFF_TC09, Zero := "Coeff".ZERO_TC09, OutValue => "Data".TC_09, Out_of_range => "Allarm".TC09_OFR)
   END_RUNG
   // the same network as SCL:
   IF "ON" THEN
       "Signal linearization"(IN0 := "ON",
                              Analog_input := "TC09":P,
                              Coeff := "Coeff".COEFF_TC09,
                              Zero := "Coeff".ZERO_TC09,
                              OutValue => "Data".TC_09,
                              Out_of_range => "Allarm".TC09_OFR);
   END_IF;
END_REGION

REGION Network 4: TC-10
   RUNG wire#powerrail
      Contact( "OFF" )
      "Signal linearization"(IN0 := "ON", Analog_input := "TC-10":P, Coeff := "Coeff".COEFF_TC10, Zero := "Coeff".ZERO_TC10, OutValue => "Data".TC_10, Out_of_range => "Allarm".TC10_OFR)
   END_RUNG
   // the same network as SCL:
   IF "OFF" THEN
       "Signal linearization"(IN0 := "ON",
                              Analog_input := "TC-10":P,
                              Coeff := "Coeff".COEFF_TC10,
                              Zero := "Coeff".ZERO_TC10,
                              OutValue => "Data".TC_10,
                              Out_of_range => "Allarm".TC10_OFR);
   END_IF;
END_REGION

REGION Network 5: CLIENT 1 BWF01 flow rate
   RUNG wire#powerrail
      Contact( "ON" )
      wire#w1
      Contact( "ON" )
      "Signal linearization"(IN0 := "ON", Analog_input := "BWF01_FlowRate":P, Coeff := "Coeff".COEFF_BWF1_FEEDER_FLOW_RATE, Zero := "Coeff".ZERO_BWF1_FEEDER_FLOW_RATE, OutValue => "Data".CLIENT_1, Out_of_range => "Allarm".Flow_rate_BWF01_OFR)
   END_RUNG
   RUNG wire#w1
      Contact( "ON" )
      wire#w2
      Contact( "BWF 01 RUN" )
      { S7_Templates := "SrcType := Int"; S7_GenerateENO := "TRUE" } Mul(in1 := "Data".SET_PERC_BWF01, in2 := "Data2".Set_TH, out => #temp4)
      { S7_Templates := "SrcType := Int"; S7_GenerateENO := "TRUE" } Div(in1 := #temp4, in2 := 100, out => "Data".CLIENT_1)
   END_RUNG
   RUNG wire#w2
      I_Contact( "BWF 01 RUN" )
      { S7_GenerateENO := "TRUE" } Move(in := 0, out1 => "Data".CLIENT_1)
   END_RUNG
   // the same network as SCL:
   // ENO of a box is taken as its EN; it also drops when the box reports an error
   #_w1 := "ON";
   IF "ON" AND "ON" THEN
       "Signal linearization"(IN0 := "ON",
                              Analog_input := "BWF01_FlowRate":P,
                              Coeff := "Coeff".COEFF_BWF1_FEEDER_FLOW_RATE,
                              Zero := "Coeff".ZERO_BWF1_FEEDER_FLOW_RATE,
                              OutValue => "Data".CLIENT_1,
                              Out_of_range => "Allarm".Flow_rate_BWF01_OFR);
   END_IF;
   #_w2 := #_w1 AND "ON";
   IF #_w2 AND "BWF 01 RUN" THEN
       #temp4 := "Data".SET_PERC_BWF01 * "Data2".Set_TH;
       "Data".CLIENT_1 := #temp4 / 100;
   END_IF;
   IF #_w2 AND NOT "BWF 01 RUN" THEN "Data".CLIENT_1 := 0; END_IF;
END_REGION

REGION Network 6: CLIENT 2 BWF02 flow rate
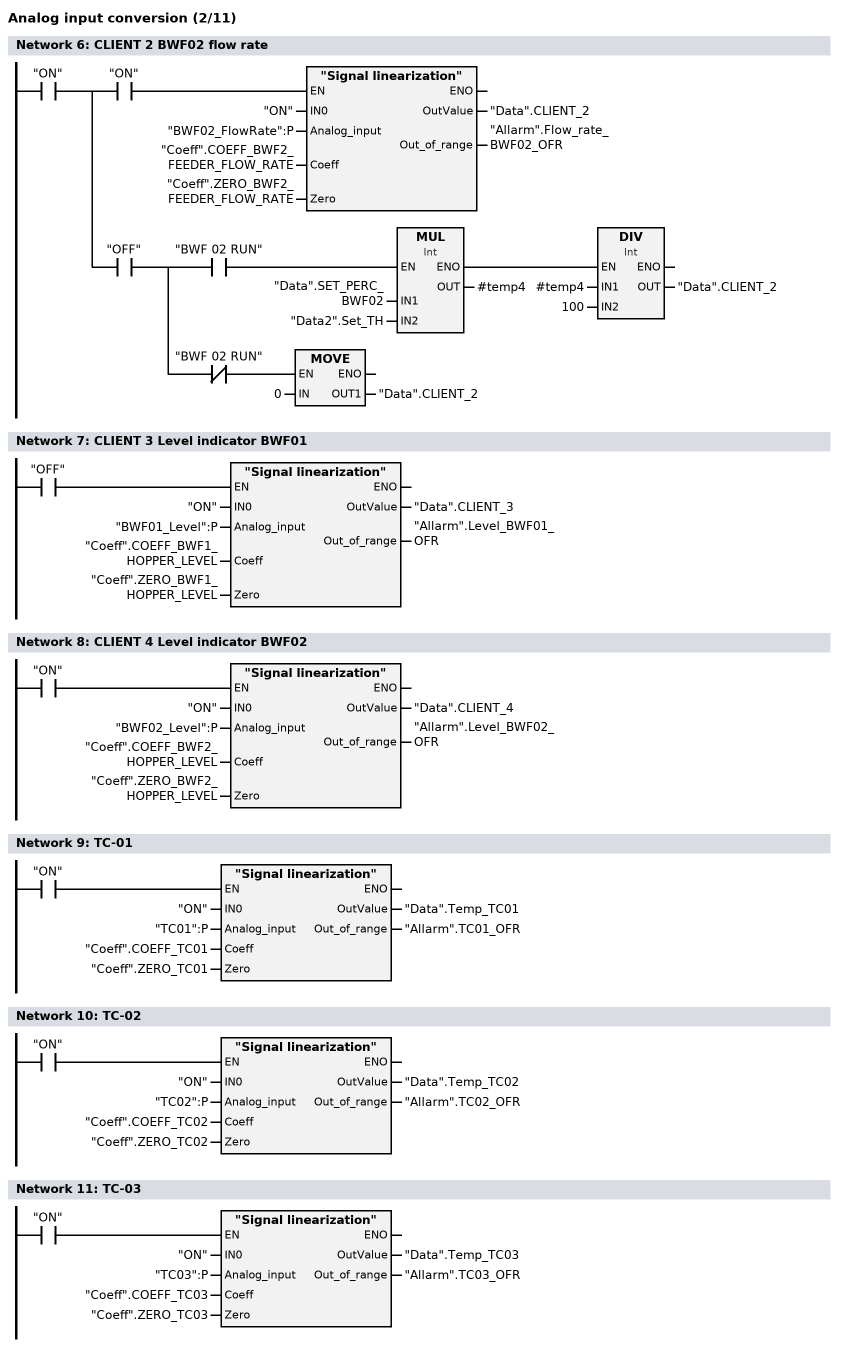
   RUNG wire#powerrail
      Contact( "ON" )
      wire#w1
      Contact( "ON" )
      "Signal linearization"(IN0 := "ON", Analog_input := "BWF02_FlowRate":P, Coeff := "Coeff".COEFF_BWF2_FEEDER_FLOW_RATE, Zero := "Coeff".ZERO_BWF2_FEEDER_FLOW_RATE, OutValue => "Data".CLIENT_2, Out_of_range => "Allarm".Flow_rate_BWF02_OFR)
   END_RUNG
   RUNG wire#w1
      Contact( "OFF" )
      wire#w2
      Contact( "BWF 02 RUN" )
      { S7_Templates := "SrcType := Int"; S7_GenerateENO := "TRUE" } Mul(in1 := "Data".SET_PERC_BWF02, in2 := "Data2".Set_TH, out => #temp4)
      { S7_Templates := "SrcType := Int"; S7_GenerateENO := "TRUE" } Div(in1 := #temp4, in2 := 100, out => "Data".CLIENT_2)
   END_RUNG
   RUNG wire#w2
      I_Contact( "BWF 02 RUN" )
      { S7_GenerateENO := "TRUE" } Move(in := 0, out1 => "Data".CLIENT_2)
   END_RUNG
   // the same network as SCL:
   // ENO of a box is taken as its EN; it also drops when the box reports an error
   #_w1 := "ON";
   IF "ON" AND "ON" THEN
       "Signal linearization"(IN0 := "ON",
                              Analog_input := "BWF02_FlowRate":P,
                              Coeff := "Coeff".COEFF_BWF2_FEEDER_FLOW_RATE,
                              Zero := "Coeff".ZERO_BWF2_FEEDER_FLOW_RATE,
                              OutValue => "Data".CLIENT_2,
                              Out_of_range => "Allarm".Flow_rate_BWF02_OFR);
   END_IF;
   #_w2 := #_w1 AND "OFF";
   IF #_w2 AND "BWF 02 RUN" THEN
       #temp4 := "Data".SET_PERC_BWF02 * "Data2".Set_TH;
       "Data".CLIENT_2 := #temp4 / 100;
   END_IF;
   IF #_w2 AND NOT "BWF 02 RUN" THEN "Data".CLIENT_2 := 0; END_IF;
END_REGION

REGION Network 7: CLIENT 3 Level indicator BWF01
   RUNG wire#powerrail
      Contact( "OFF" )
      "Signal linearization"(IN0 := "ON", Analog_input := "BWF01_Level":P, Coeff := "Coeff".COEFF_BWF1_HOPPER_LEVEL, Zero := "Coeff".ZERO_BWF1_HOPPER_LEVEL, OutValue => "Data".CLIENT_3, Out_of_range => "Allarm".Level_BWF01_OFR)
   END_RUNG
   // the same network as SCL:
   IF "OFF" THEN
       "Signal linearization"(IN0 := "ON",
                              Analog_input := "BWF01_Level":P,
                              Coeff := "Coeff".COEFF_BWF1_HOPPER_LEVEL,
                              Zero := "Coeff".ZERO_BWF1_HOPPER_LEVEL,
                              OutValue => "Data".CLIENT_3,
                              Out_of_range => "Allarm".Level_BWF01_OFR);
   END_IF;
END_REGION

REGION Network 8: CLIENT 4 Level indicator BWF02
   RUNG wire#powerrail
      Contact( "ON" )
      "Signal linearization"(IN0 := "ON", Analog_input := "BWF02_Level":P, Coeff := "Coeff".COEFF_BWF2_HOPPER_LEVEL, Zero := "Coeff".ZERO_BWF2_HOPPER_LEVEL, OutValue => "Data".CLIENT_4, Out_of_range => "Allarm".Level_BWF02_OFR)
   END_RUNG
   // the same network as SCL:
   IF "ON" THEN
       "Signal linearization"(IN0 := "ON",
                              Analog_input := "BWF02_Level":P,
                              Coeff := "Coeff".COEFF_BWF2_HOPPER_LEVEL,
                              Zero := "Coeff".ZERO_BWF2_HOPPER_LEVEL,
                              OutValue => "Data".CLIENT_4,
                              Out_of_range => "Allarm".Level_BWF02_OFR);
   END_IF;
END_REGION

REGION Network 9: TC-01
   RUNG wire#powerrail
      Contact( "ON" )
      "Signal linearization"(IN0 := "ON", Analog_input := "TC01":P, Coeff := "Coeff".COEFF_TC01, Zero := "Coeff".ZERO_TC01, OutValue => "Data".Temp_TC01, Out_of_range => "Allarm".TC01_OFR)
   END_RUNG
   // the same network as SCL:
   IF "ON" THEN
       "Signal linearization"(IN0 := "ON",
                              Analog_input := "TC01":P,
                              Coeff := "Coeff".COEFF_TC01,
                              Zero := "Coeff".ZERO_TC01,
                              OutValue => "Data".Temp_TC01,
                              Out_of_range => "Allarm".TC01_OFR);
   END_IF;
END_REGION

REGION Network 10: TC-02
   RUNG wire#powerrail
      Contact( "ON" )
      "Signal linearization"(IN0 := "ON", Analog_input := "TC02":P, Coeff := "Coeff".COEFF_TC02, Zero := "Coeff".ZERO_TC02, OutValue => "Data".Temp_TC02, Out_of_range => "Allarm".TC02_OFR)
   END_RUNG
   // the same network as SCL:
   IF "ON" THEN
       "Signal linearization"(IN0 := "ON",
                              Analog_input := "TC02":P,
                              Coeff := "Coeff".COEFF_TC02,
                              Zero := "Coeff".ZERO_TC02,
                              OutValue => "Data".Temp_TC02,
                              Out_of_range => "Allarm".TC02_OFR);
   END_IF;
END_REGION

REGION Network 11: TC-03
   RUNG wire#powerrail
      Contact( "ON" )
      "Signal linearization"(IN0 := "ON", Analog_input := "TC03":P, Coeff := "Coeff".COEFF_TC03, Zero := "Coeff".ZERO_TC03, OutValue => "Data".Temp_TC03, Out_of_range => "Allarm".TC03_OFR)
   END_RUNG
   // the same network as SCL:
   IF "ON" THEN
       "Signal linearization"(IN0 := "ON",
                              Analog_input := "TC03":P,
                              Coeff := "Coeff".COEFF_TC03,
                              Zero := "Coeff".ZERO_TC03,
                              OutValue => "Data".Temp_TC03,
                              Out_of_range => "Allarm".TC03_OFR);
   END_IF;
END_REGION

REGION Network 12: TC-06
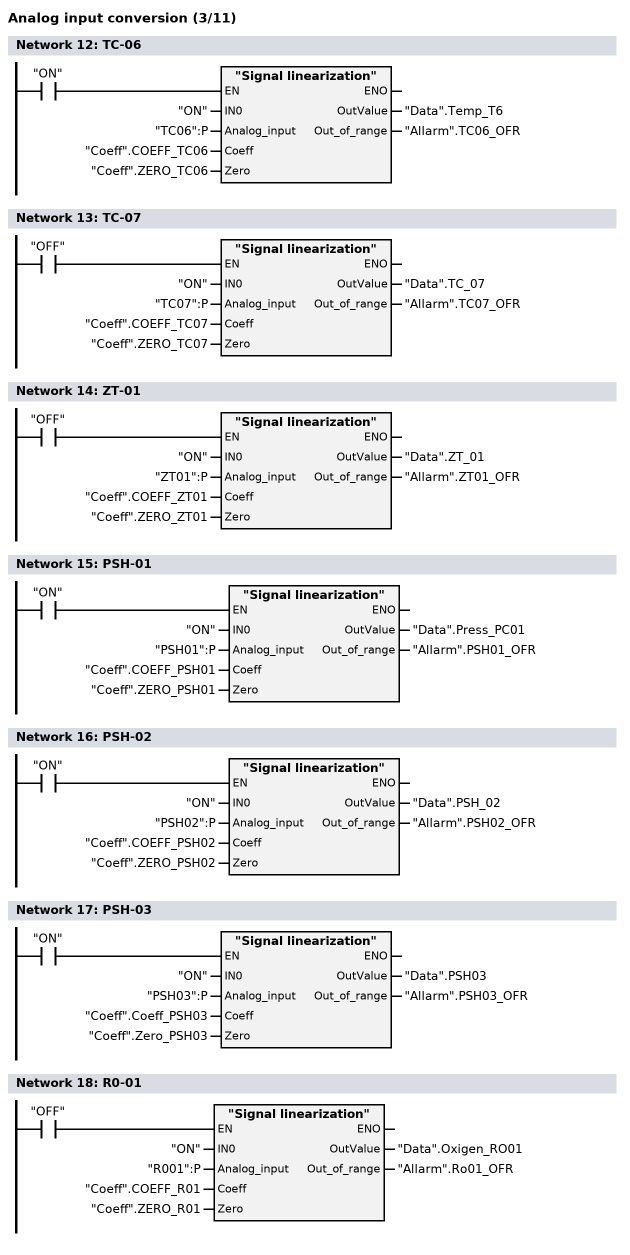
   RUNG wire#powerrail
      Contact( "ON" )
      "Signal linearization"(IN0 := "ON", Analog_input := "TC06":P, Coeff := "Coeff".COEFF_TC06, Zero := "Coeff".ZERO_TC06, OutValue => "Data".Temp_T6, Out_of_range => "Allarm".TC06_OFR)
   END_RUNG
   // the same network as SCL:
   IF "ON" THEN
       "Signal linearization"(IN0 := "ON",
                              Analog_input := "TC06":P,
                              Coeff := "Coeff".COEFF_TC06,
                              Zero := "Coeff".ZERO_TC06,
                              OutValue => "Data".Temp_T6,
                              Out_of_range => "Allarm".TC06_OFR);
   END_IF;
END_REGION

REGION Network 13: TC-07
   RUNG wire#powerrail
      Contact( "OFF" )
      "Signal linearization"(IN0 := "ON", Analog_input := "TC07":P, Coeff := "Coeff".COEFF_TC07, Zero := "Coeff".ZERO_TC07, OutValue => "Data".TC_07, Out_of_range => "Allarm".TC07_OFR)
   END_RUNG
   // the same network as SCL:
   IF "OFF" THEN
       "Signal linearization"(IN0 := "ON",
                              Analog_input := "TC07":P,
                              Coeff := "Coeff".COEFF_TC07,
                              Zero := "Coeff".ZERO_TC07,
                              OutValue => "Data".TC_07,
                              Out_of_range => "Allarm".TC07_OFR);
   END_IF;
END_REGION

REGION Network 14: ZT-01
   RUNG wire#powerrail
      Contact( "OFF" )
      "Signal linearization"(IN0 := "ON", Analog_input := "ZT01":P, Coeff := "Coeff".COEFF_ZT01, Zero := "Coeff".ZERO_ZT01, OutValue => "Data".ZT_01, Out_of_range => "Allarm".ZT01_OFR)
   END_RUNG
   // the same network as SCL:
   IF "OFF" THEN
       "Signal linearization"(IN0 := "ON",
                              Analog_input := "ZT01":P,
                              Coeff := "Coeff".COEFF_ZT01,
                              Zero := "Coeff".ZERO_ZT01,
                              OutValue => "Data".ZT_01,
                              Out_of_range => "Allarm".ZT01_OFR);
   END_IF;
END_REGION

REGION Network 15: PSH-01
   RUNG wire#powerrail
      Contact( "ON" )
      "Signal linearization"(IN0 := "ON", Analog_input := "PSH01":P, Coeff := "Coeff".COEFF_PSH01, Zero := "Coeff".ZERO_PSH01, OutValue => "Data".Press_PC01, Out_of_range => "Allarm".PSH01_OFR)
   END_RUNG
   // the same network as SCL:
   IF "ON" THEN
       "Signal linearization"(IN0 := "ON",
                              Analog_input := "PSH01":P,
                              Coeff := "Coeff".COEFF_PSH01,
                              Zero := "Coeff".ZERO_PSH01,
                              OutValue => "Data".Press_PC01,
                              Out_of_range => "Allarm".PSH01_OFR);
   END_IF;
END_REGION

REGION Network 16: PSH-02
   RUNG wire#powerrail
      Contact( "ON" )
      "Signal linearization"(IN0 := "ON", Analog_input := "PSH02":P, Coeff := "Coeff".COEFF_PSH02, Zero := "Coeff".ZERO_PSH02, OutValue => "Data".PSH_02, Out_of_range => "Allarm".PSH02_OFR)
   END_RUNG
   // the same network as SCL:
   IF "ON" THEN
       "Signal linearization"(IN0 := "ON",
                              Analog_input := "PSH02":P,
                              Coeff := "Coeff".COEFF_PSH02,
                              Zero := "Coeff".ZERO_PSH02,
                              OutValue => "Data".PSH_02,
                              Out_of_range => "Allarm".PSH02_OFR);
   END_IF;
END_REGION

REGION Network 17: PSH-03
   RUNG wire#powerrail
      Contact( "ON" )
      "Signal linearization"(IN0 := "ON", Analog_input := "PSH03":P, Coeff := "Coeff".Coeff_PSH03, Zero := "Coeff".Zero_PSH03, OutValue => "Data".PSH03, Out_of_range => "Allarm".PSH03_OFR)
   END_RUNG
   // the same network as SCL:
   IF "ON" THEN
       "Signal linearization"(IN0 := "ON",
                              Analog_input := "PSH03":P,
                              Coeff := "Coeff".Coeff_PSH03,
                              Zero := "Coeff".Zero_PSH03,
                              OutValue => "Data".PSH03,
                              Out_of_range => "Allarm".PSH03_OFR);
   END_IF;
END_REGION

REGION Network 18: R0-01
   RUNG wire#powerrail
      Contact( "OFF" )
      "Signal linearization"(IN0 := "ON", Analog_input := "R001":P, Coeff := "Coeff".COEFF_R01, Zero := "Coeff".ZERO_R01, OutValue => "Data".Oxigen_RO01, Out_of_range => "Allarm".Ro01_OFR)
   END_RUNG
   // the same network as SCL:
   IF "OFF" THEN
       "Signal linearization"(IN0 := "ON",
                              Analog_input := "R001":P,
                              Coeff := "Coeff".COEFF_R01,
                              Zero := "Coeff".ZERO_R01,
                              OutValue => "Data".Oxigen_RO01,
                              Out_of_range => "Allarm".Ro01_OFR);
   END_IF;
END_REGION

REGION Network 19: R0-02
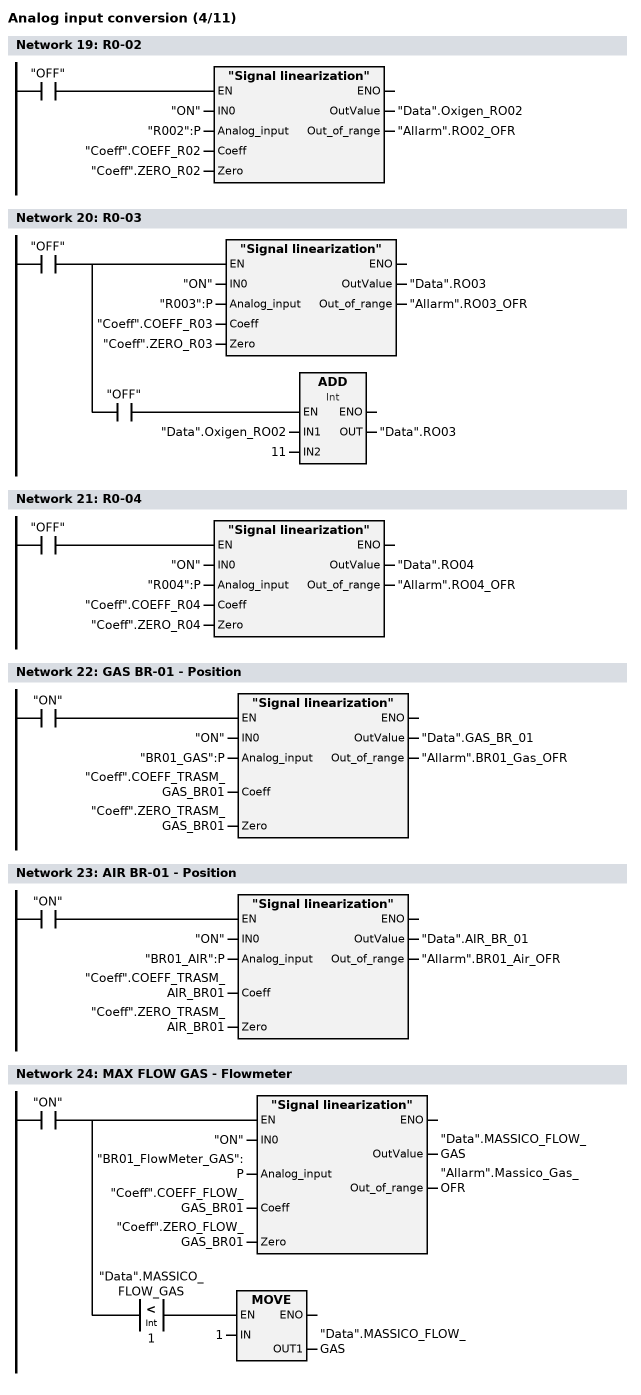
   RUNG wire#powerrail
      Contact( "OFF" )
      "Signal linearization"(IN0 := "ON", Analog_input := "R002":P, Coeff := "Coeff".COEFF_R02, Zero := "Coeff".ZERO_R02, OutValue => "Data".Oxigen_RO02, Out_of_range => "Allarm".RO02_OFR)
   END_RUNG
   // the same network as SCL:
   IF "OFF" THEN
       "Signal linearization"(IN0 := "ON",
                              Analog_input := "R002":P,
                              Coeff := "Coeff".COEFF_R02,
                              Zero := "Coeff".ZERO_R02,
                              OutValue => "Data".Oxigen_RO02,
                              Out_of_range => "Allarm".RO02_OFR);
   END_IF;
END_REGION

REGION Network 20: R0-03
   RUNG wire#powerrail
      Contact( "OFF" )
      wire#w1
      "Signal linearization"(IN0 := "ON", Analog_input := "R003":P, Coeff := "Coeff".COEFF_R03, Zero := "Coeff".ZERO_R03, OutValue => "Data".RO03, Out_of_range => "Allarm".RO03_OFR)
   END_RUNG
   RUNG wire#w1
      Contact( "OFF" )
      { S7_Templates := "SrcType := Int"; S7_GenerateENO := "TRUE" } Add(in1 := "Data".Oxigen_RO02, in2 := 11, out => "Data".RO03)
   END_RUNG
   // the same network as SCL:
   #_w1 := "OFF";
   IF #_w1 THEN
       "Signal linearization"(IN0 := "ON",
                              Analog_input := "R003":P,
                              Coeff := "Coeff".COEFF_R03,
                              Zero := "Coeff".ZERO_R03,
                              OutValue => "Data".RO03,
                              Out_of_range => "Allarm".RO03_OFR);
   END_IF;
   IF #_w1 AND "OFF" THEN "Data".RO03 := "Data".Oxigen_RO02 + 11; END_IF;
END_REGION

REGION Network 21: R0-04
   RUNG wire#powerrail
      Contact( "OFF" )
      "Signal linearization"(IN0 := "ON", Analog_input := "R004":P, Coeff := "Coeff".COEFF_R04, Zero := "Coeff".ZERO_R04, OutValue => "Data".RO04, Out_of_range => "Allarm".RO04_OFR)
   END_RUNG
   // the same network as SCL:
   IF "OFF" THEN
       "Signal linearization"(IN0 := "ON",
                              Analog_input := "R004":P,
                              Coeff := "Coeff".COEFF_R04,
                              Zero := "Coeff".ZERO_R04,
                              OutValue => "Data".RO04,
                              Out_of_range => "Allarm".RO04_OFR);
   END_IF;
END_REGION

REGION Network 22: GAS BR-01 - Position
   RUNG wire#powerrail
      Contact( "ON" )
      "Signal linearization"(IN0 := "ON", Analog_input := "BR01_GAS":P, Coeff := "Coeff".COEFF_TRASM_GAS_BR01, Zero := "Coeff".ZERO_TRASM_GAS_BR01, OutValue => "Data".GAS_BR_01, Out_of_range => "Allarm".BR01_Gas_OFR)
   END_RUNG
   // the same network as SCL:
   IF "ON" THEN
       "Signal linearization"(IN0 := "ON",
                              Analog_input := "BR01_GAS":P,
                              Coeff := "Coeff".COEFF_TRASM_GAS_BR01,
                              Zero := "Coeff".ZERO_TRASM_GAS_BR01,
                              OutValue => "Data".GAS_BR_01,
                              Out_of_range => "Allarm".BR01_Gas_OFR);
   END_IF;
END_REGION

REGION Network 23: AIR BR-01 - Position
   RUNG wire#powerrail
      Contact( "ON" )
      "Signal linearization"(IN0 := "ON", Analog_input := "BR01_AIR":P, Coeff := "Coeff".COEFF_TRASM_AIR_BR01, Zero := "Coeff".ZERO_TRASM_AIR_BR01, OutValue => "Data".AIR_BR_01, Out_of_range => "Allarm".BR01_Air_OFR)
   END_RUNG
   // the same network as SCL:
   IF "ON" THEN
       "Signal linearization"(IN0 := "ON",
                              Analog_input := "BR01_AIR":P,
                              Coeff := "Coeff".COEFF_TRASM_AIR_BR01,
                              Zero := "Coeff".ZERO_TRASM_AIR_BR01,
                              OutValue => "Data".AIR_BR_01,
                              Out_of_range => "Allarm".BR01_Air_OFR);
   END_IF;
END_REGION

REGION Network 24: MAX FLOW GAS - Flowmeter
   RUNG wire#powerrail
      Contact( "ON" )
      wire#w1
      "Signal linearization"(IN0 := "ON", Analog_input := "BR01_FlowMeter_GAS":P, Coeff := "Coeff".COEFF_FLOW_GAS_BR01, Zero := "Coeff".ZERO_FLOW_GAS_BR01, OutValue => "Data".MASSICO_FLOW_GAS, Out_of_range => "Allarm".Massico_Gas_OFR)
   END_RUNG
   RUNG wire#w1
      { S7_Templates := "SrcType := Int" } LT_Contact(in1 := "Data".MASSICO_FLOW_GAS, in2 := 1)
      { S7_GenerateENO := "TRUE" } Move(in := 1, out1 => "Data".MASSICO_FLOW_GAS)
   END_RUNG
   // the same network as SCL:
   #_w1 := "ON";
   IF #_w1 THEN
       "Signal linearization"(IN0 := "ON",
                              Analog_input := "BR01_FlowMeter_GAS":P,
                              Coeff := "Coeff".COEFF_FLOW_GAS_BR01,
                              Zero := "Coeff".ZERO_FLOW_GAS_BR01,
                              OutValue => "Data".MASSICO_FLOW_GAS,
                              Out_of_range => "Allarm".Massico_Gas_OFR);
   END_IF;
   IF #_w1 AND ("Data".MASSICO_FLOW_GAS < 1) THEN "Data".MASSICO_FLOW_GAS := 1; END_IF;
END_REGION

REGION Network 25: MAX FLOW AIR - Flowmeter
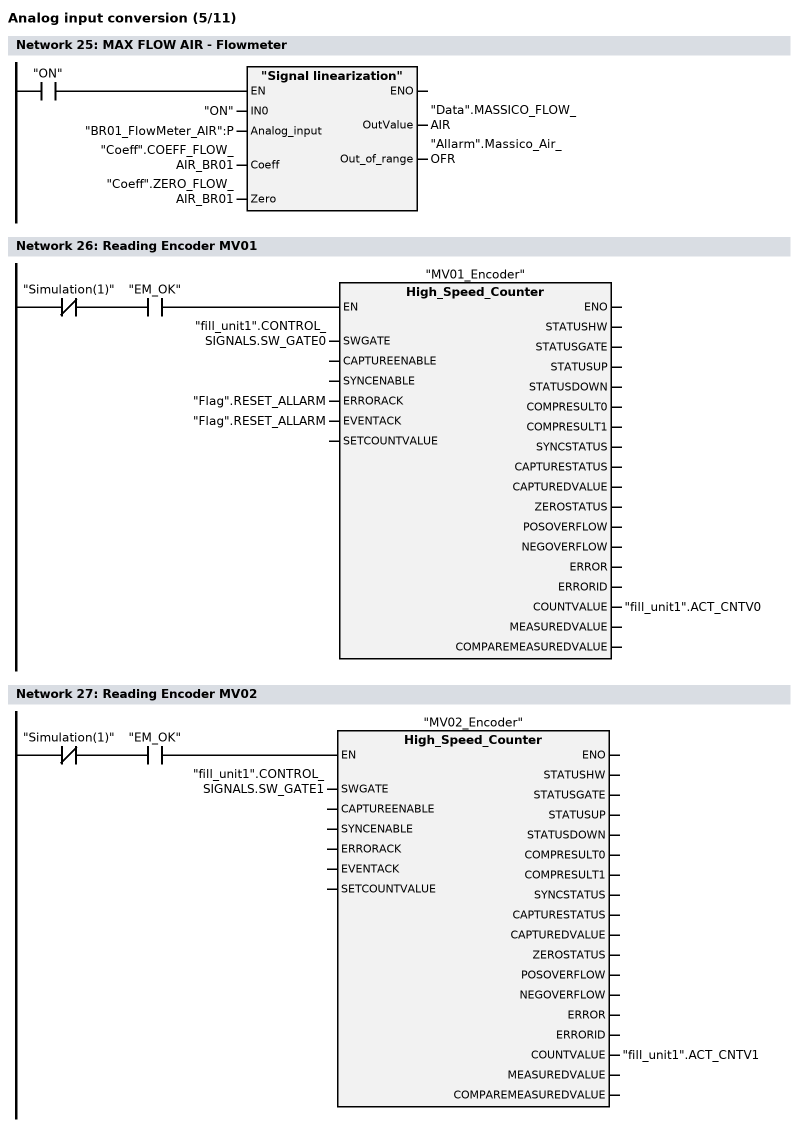
   RUNG wire#powerrail
      Contact( "ON" )
      "Signal linearization"(IN0 := "ON", Analog_input := "BR01_FlowMeter_AIR":P, Coeff := "Coeff".COEFF_FLOW_AIR_BR01, Zero := "Coeff".ZERO_FLOW_AIR_BR01, OutValue => "Data".MASSICO_FLOW_AIR, Out_of_range => "Allarm".Massico_Air_OFR)
   END_RUNG
   // the same network as SCL:
   IF "ON" THEN
       "Signal linearization"(IN0 := "ON",
                              Analog_input := "BR01_FlowMeter_AIR":P,
                              Coeff := "Coeff".COEFF_FLOW_AIR_BR01,
                              Zero := "Coeff".ZERO_FLOW_AIR_BR01,
                              OutValue => "Data".MASSICO_FLOW_AIR,
                              Out_of_range => "Allarm".Massico_Air_OFR);
   END_IF;
END_REGION

REGION Network 26: Reading Encoder MV01
   IF NOT "Simulation(1)" AND "EM_OK" THEN
       "MV01_Encoder"(SwGate := "fill_unit1".CONTROL_SIGNALS.SW_GATE0,   // High_Speed_Counter
                      ErrorAck := "Flag".RESET_ALLARM,
                      EventAck := "Flag".RESET_ALLARM,
                      CountValue => "fill_unit1".ACT_CNTV0);
   END_IF;
END_REGION

REGION Network 27: Reading Encoder MV02
   IF NOT "Simulation(1)" AND "EM_OK" THEN
       "MV02_Encoder"(SwGate := "fill_unit1".CONTROL_SIGNALS.SW_GATE1, CountValue => "fill_unit1".ACT_CNTV1);   // High_Speed_Counter
   END_IF;
END_REGION

REGION Network 28: Reading Encoder MV03
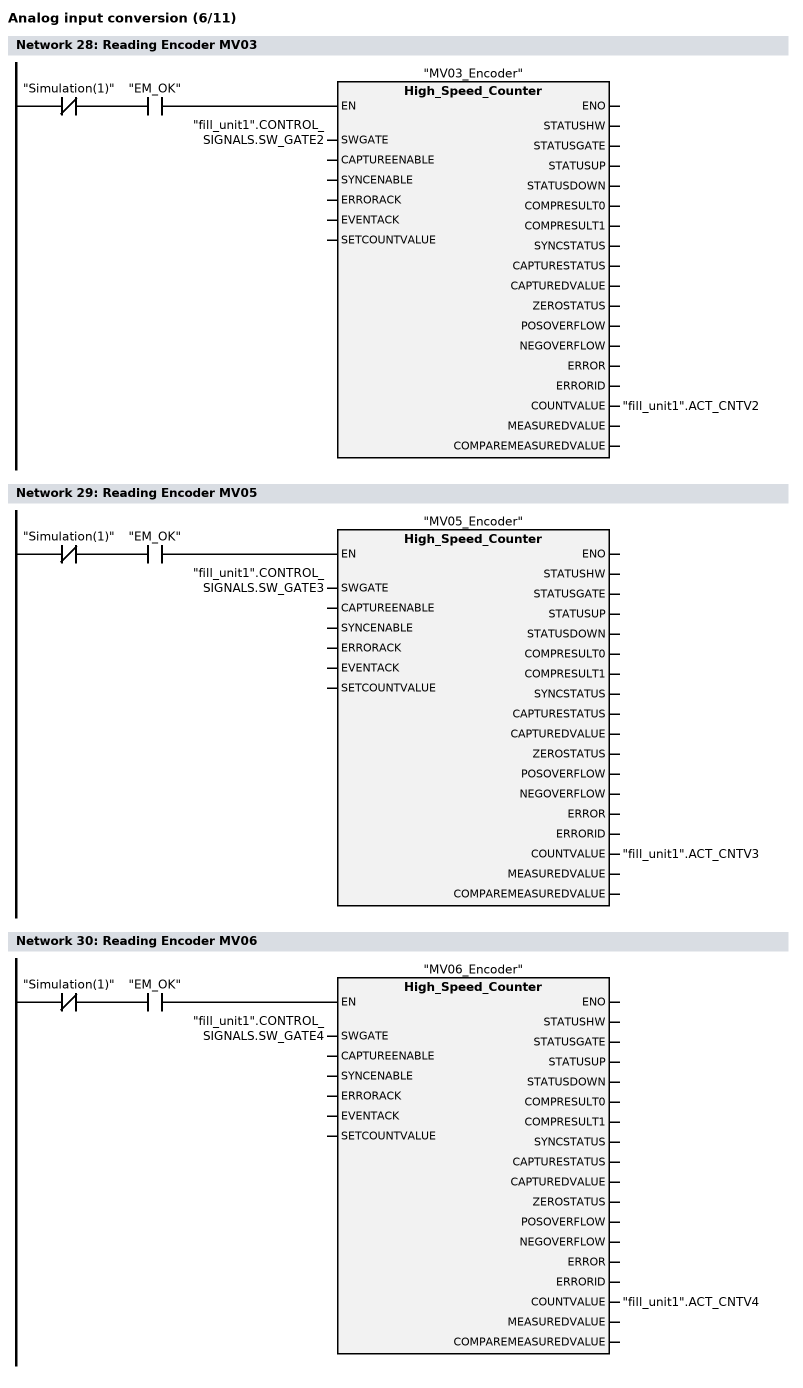
   IF NOT "Simulation(1)" AND "EM_OK" THEN
       "MV03_Encoder"(SwGate := "fill_unit1".CONTROL_SIGNALS.SW_GATE2, CountValue => "fill_unit1".ACT_CNTV2);   // High_Speed_Counter
   END_IF;
END_REGION

REGION Network 29: Reading Encoder MV05
   IF NOT "Simulation(1)" AND "EM_OK" THEN
       "MV05_Encoder"(SwGate := "fill_unit1".CONTROL_SIGNALS.SW_GATE3, CountValue => "fill_unit1".ACT_CNTV3);   // High_Speed_Counter
   END_IF;
END_REGION

REGION Network 30: Reading Encoder MV06
   IF NOT "Simulation(1)" AND "EM_OK" THEN
       "MV06_Encoder"(SwGate := "fill_unit1".CONTROL_SIGNALS.SW_GATE4, CountValue => "fill_unit1".ACT_CNTV4);   // High_Speed_Counter
   END_IF;
END_REGION

REGION Network 31: Store current position value at power-off
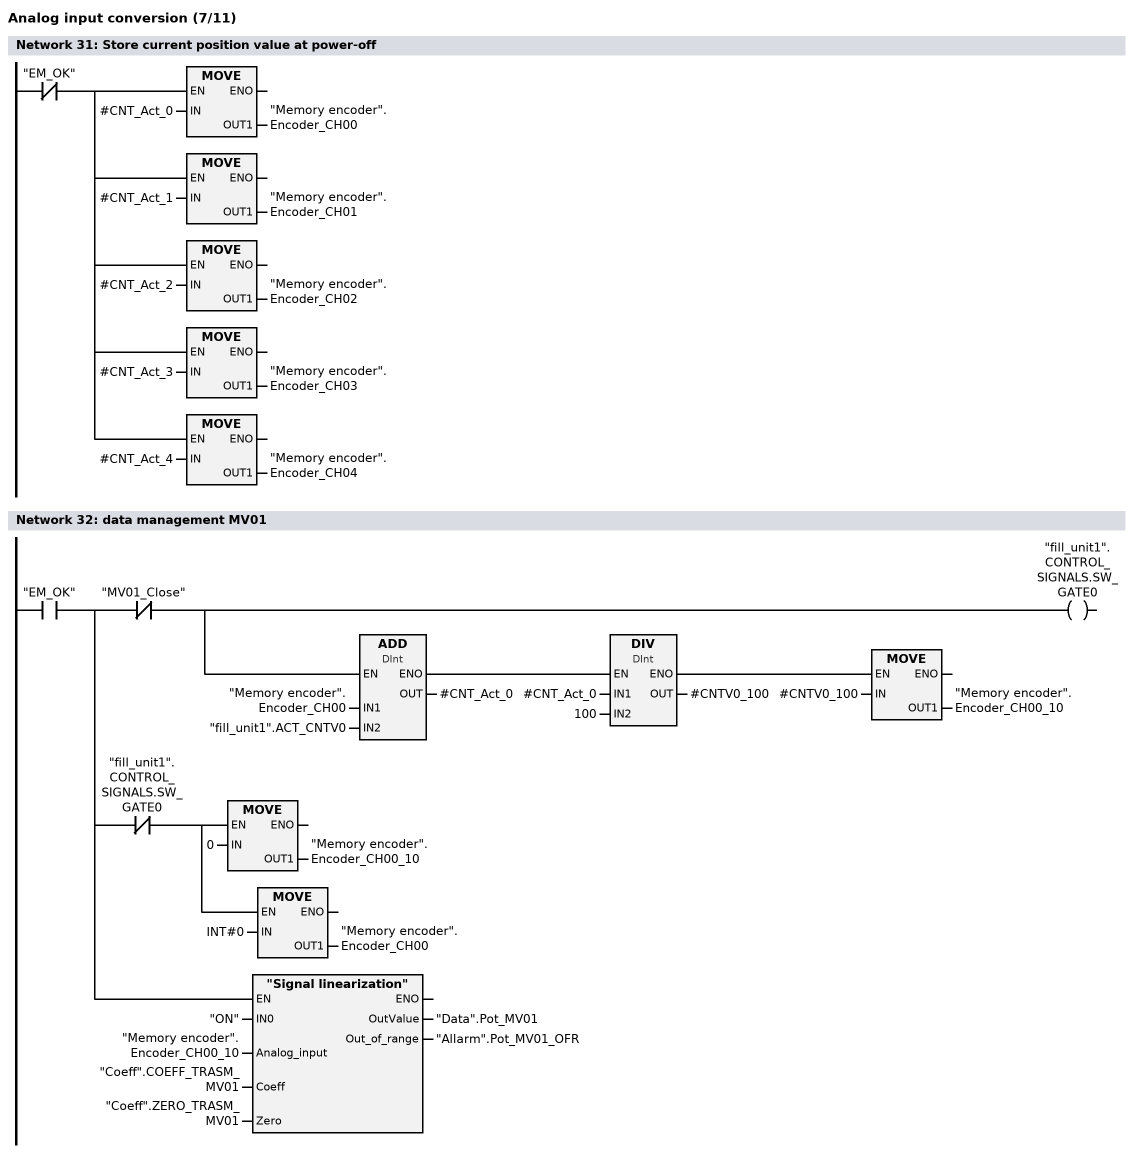
   RUNG wire#powerrail
      I_Contact( "EM_OK" )
      wire#w1
      { S7_GenerateENO := "TRUE" } Move(in := #CNT_Act_0, out1 => "Memory encoder".Encoder_CH00)
   END_RUNG
   RUNG wire#w1
      { S7_GenerateENO := "TRUE" } Move(in := #CNT_Act_1, out1 => "Memory encoder".Encoder_CH01)
   END_RUNG
   RUNG wire#w1
      { S7_GenerateENO := "TRUE" } Move(in := #CNT_Act_2, out1 => "Memory encoder".Encoder_CH02)
   END_RUNG
   RUNG wire#w1
      { S7_GenerateENO := "TRUE" } Move(in := #CNT_Act_3, out1 => "Memory encoder".Encoder_CH03)
   END_RUNG
   RUNG wire#w1
      { S7_GenerateENO := "TRUE" } Move(in := #CNT_Act_4, out1 => "Memory encoder".Encoder_CH04)
   END_RUNG
   // the same network as SCL:
   IF NOT "EM_OK" THEN
       "Memory encoder".Encoder_CH00 := #CNT_Act_0;
       "Memory encoder".Encoder_CH01 := #CNT_Act_1;
       "Memory encoder".Encoder_CH02 := #CNT_Act_2;
       "Memory encoder".Encoder_CH03 := #CNT_Act_3;
       "Memory encoder".Encoder_CH04 := #CNT_Act_4;
   END_IF;
END_REGION

